LIN {X 0,Y 339.06,Z 977.216,A -85,B 0,C 180,E1 15201.009,E2 15201.009} C_VEL
LIN {X 0,Y 338.438,Z 981.844,A -85,B 0,C 180,E1 15198.238,E2 15198.238} C_VEL
LIN {X 0,Y 338.121,Z 984.855,A -85,B 0,C 180,E1 15195.268,E2 15195.268} C_VEL
LIN {X 0,Y 338.142,Z 986.085,A -85,B 0,C 180,E1 15192.269,E2 15192.269} C_VEL
LIN {X 0,Y 338.465,Z 985.515,A -85,B 0,C 180,E1 15189.419,E2 15189.419} C_VEL
LIN {X 0,Y 339.2,Z 983.049,A -85,B 0,C 180,E1 15186.367,E2 15186.367} C_VEL
LIN {X 0,Y 340.341,Z 978.866,A -85,B 0,C 180,E1 15183.478,E2 15183.478} C_VEL
LIN {X 0,Y 341.875,Z 973.019,A -85,B 0,C 180,E1 15180.764,E2 15180.764} C_VEL
LIN {X 0,Y 343.946,Z 965.145,A -85,B 0,C 180,E1 15178.057,E2 15178.057} C_VEL
LIN {X 0,Y 346.224,Z 956.156,A -85,B 0,C 180,E1 15175.685,E2 15175.685} C_VEL
LIN {X 0,Y 348.825,Z 945.138,A -85,B 0,C 180,E1 15173.402,E2 15173.402} C_VEL
LIN {X 0,Y 351.492,Z 932.886,A -85,B 0,C 180,E1 15171.379,E2 15171.379} C_VEL
LIN {X 0,Y 353.963,Z 920.077,A -85,B 0,C 180,E1 15169.694,E2 15169.694} C_VEL
LIN {X 0,Y 356.266,Z 906.077,A -85,B 0,C 180,E1 15168.227,E2 15168.227} C_VEL
LIN {X 0,Y 358.353,Z 890.745,A -85,B 0,C 180,E1 15166.972,E2 15166.972} C_VEL
LIN {X 0,Y 360,Z 874.678,A -85,B 0,C 180,E1 15165.985,E2 15165.985} C_VEL
LIN {X 0,Y 361.102,Z 857.67,A -85,B 0,C 180,E1 15165.259,E2 15165.259} C_VEL
LIN {X 0,Y 361.863,Z 835.3,A -85,B 0,C 180,E1 15164.69,E2 15164.69} C_VEL
LIN {X 0,Y 365.466,Z 734.296,A -85,B 0,C 180,E1 15162.572,E2 15162.572} C_VEL
LIN {X 0,Y 359.291,Z 705.714,A -85,B 0,C 180,E1 15161.014,E2 15161.014} C_VEL
LIN {X 0,Y 357.272,Z 697.189,A -85,B 0,C 180,E1 15160.487,E2 15160.487} C_VEL
LIN {X 0,Y 358.03,Z 691.708,A -85,B 0,C 180,E1 15159.549,E2 15159.549} C_VEL
LIN {X 0,Y 354.94,Z 678.848,A -85,B 0,C 180,E1 15156.327,E2 15156.327} C_VEL
LIN {X 0,Y 351.349,Z 666.673,A -85,B 0,C 180,E1 15152.913,E2 15152.913} C_VEL
LIN {X 0,Y 347.723,Z 656.229,A -85,B 0,C 180,E1 15149.642,E2 15149.642} C_VEL
LIN {X 0,Y 344.373,Z 647.376,A -85,B 0,C 180,E1 15146.56,E2 15146.56} C_VEL
LIN {X 0,Y 341.041,Z 639.591,A -85,B 0,C 180,E1 15143.499,E2 15143.499} C_VEL
LIN {X 0,Y 339.313,Z 635.632,A -85,B 0,C 180,E1 15141.795,E2 15141.795} C_VEL
LIN {X 0,Y 338.001,Z 632.231,A -85,B 0,C 180,E1 15140.157,E2 15140.157} C_VEL
LIN {X 0,Y 337.989,Z 632.124,A -85,B 0,C 180,E1 15135.793,E2 15135.793} C_VEL
LIN {X 0,Y 337.983,Z 632.122,A -85,B 0,C 180,E1 15131.432,E2 15131.432} C_VEL
LIN {X 0,Y 337.983,Z 632.127,A -85,B 0,C 180,E1 15127.138,E2 15127.138} C_VEL
LIN {X 0,Y 337.978,Z 632.134,A -85,B 0,C 180,E1 15122.713,E2 15122.713} C_VEL
LIN {X 0,Y 337.978,Z 632.135,A -85,B 0,C 180,E1 15118.475,E2 15118.475} C_VEL
LIN {X 0,Y 337.98,Z 632.122,A -85,B 0,C 180,E1 15114.057,E2 15114.057} C_VEL
LIN {X 0,Y 337.978,Z 632.112,A -85,B 0,C 180,E1 15109.776,E2 15109.776} C_VEL
LIN {X 0,Y 337.987,Z 632.108,A -85,B 0,C 180,E1 15105.437,E2 15105.437} C_VEL
LIN {X 0,Y 337.984,Z 632.108,A -85,B 0,C 180,E1 15101.189,E2 15101.189} C_VEL
LIN {X 0,Y 337.988,Z 632.11,A -85,B 0,C 180,E1 15096.928,E2 15096.928} C_VEL
LIN {X 0,Y 337.99,Z 632.112,A -85,B 0,C 180,E1 15092.557,E2 15092.557} C_VEL
LIN {X 0,Y 338.011,Z 632.35,A -85,B 0,C 180,E1 15088.825,E2 15088.825} C_VEL
LIN {X 0,Y 339.689,Z 636.177,A -85,B 0,C 180,E1 15087.208,E2 15087.208} C_VEL
LIN {X 0,Y 342.604,Z 642.181,A -85,B 0,C 180,E1 15084.906,E2 15084.906} C_VEL
LIN {X 0,Y 346.288,Z 649.982,A -85,B 0,C 180,E1 15082.257,E2 15082.257} C_VEL
LIN {X 0,Y 351.256,Z 661.463,A -85,B 0,C 180,E1 15078.887,E2 15078.887} C_VEL
LIN {X 0,Y 356.257,Z 674.185,A -85,B 0,C 180,E1 15075.667,E2 15075.667} C_VEL
LIN {X 0,Y 360.952,Z 687.923,A -85,B 0,C 180,E1 15072.655,E2 15072.655} C_VEL
LIN {X 0,Y 363.777,Z 697.683,A -85,B 0,C 180,E1 15070.762,E2 15070.762} C_VEL
LIN {X 0,Y 362.254,Z 706.393,A -85,B 0,C 180,E1 15069.715,E2 15069.715} C_VEL
LIN {X 0,Y 366.045,Z 739.38,A -85,B 0,C 180,E1 15068.36,E2 15068.36} C_VEL
LIN {X 0,Y 366.683,Z 749.229,A -85,B 0,C 180,E1 15068.034,E2 15068.034} C_VEL
LIN {X 0,Y 361.071,Z 910.999,A -85,B 0,C 180,E1 15064.714,E2 15064.714} C_VEL
LIN {X 0,Y 359.486,Z 930.013,A -85,B 0,C 180,E1 15064.068,E2 15064.068} C_VEL
LIN {X 0,Y 357.3,Z 948.27,A -85,B 0,C 180,E1 15063.167,E2 15063.167} C_VEL
LIN {X 0,Y 354.735,Z 965.817,A -85,B 0,C 180,E1 15061.998,E2 15061.998} C_VEL
LIN {X 0,Y 351.945,Z 982.563,A -85,B 0,C 180,E1 15060.566,E2 15060.566} C_VEL
LIN {X 0,Y 348.905,Z 999.229,A -85,B 0,C 180,E1 15058.779,E2 15058.779} C_VEL
LIN {X 0,Y 345.971,Z 1014.591,A -85,B 0,C 180,E1 15056.746,E2 15056.746} C_VEL
LIN {X 0,Y 343.233,Z 1028.904,A -85,B 0,C 180,E1 15054.434,E2 15054.434} C_VEL
LIN {X 0,Y 340.862,Z 1041.948,A -85,B 0,C 180,E1 15051.871,E2 15051.871} C_VEL
LIN {X 0,Y 338.983,Z 1053.504,A -85,B 0,C 180,E1 15049.111,E2 15049.111} C_VEL
LIN {X 0,Y 337.683,Z 1063.577,A -85,B 0,C 180,E1 15046.16,E2 15046.16} C_VEL
LIN {X 0,Y 336.936,Z 1072.093,A -85,B 0,C 180,E1 15043.034,E2 15043.034} C_VEL
LIN {X 0,Y 336.742,Z 1078.623,A -85,B 0,C 180,E1 15039.916,E2 15039.916} C_VEL
LIN {X 0,Y 336.869,Z 1083.303,A -85,B 0,C 180,E1 15036.818,E2 15036.818} C_VEL
LIN {X 0,Y 337.128,Z 1086.084,A -85,B 0,C 180,E1 15033.911,E2 15033.911} C_VEL
LIN {X 0,Y 337.307,Z 1087.318,A -85,B 0,C 180,E1 15031.019,E2 15031.019} C_VEL
LIN {X 0,Y 337.291,Z 1086.995,A -85,B 0,C 180,E1 15028.131,E2 15028.131} C_VEL
LIN {X 0,Y 337.092,Z 1085.098,A -85,B 0,C 180,E1 15025.236,E2 15025.236} C_VEL
LIN {X 0,Y 336.876,Z 1081.6,A -85,B 0,C 180,E1 15022.324,E2 15022.324} C_VEL
LIN {X 0,Y 336.836,Z 1076.055,A -85,B 0,C 180,E1 15019.221,E2 15019.221} C_VEL
LIN {X 0,Y 337.123,Z 1068.997,A -85,B 0,C 180,E1 15016.274,E2 15016.274} C_VEL
LIN {X 0,Y 337.906,Z 1059.968,A -85,B 0,C 180,E1 15013.32,E2 15013.32} C_VEL
LIN {X 0,Y 339.17,Z 1049.43,A -85,B 0,C 180,E1 15010.541,E2 15010.541} C_VEL
LIN {X 0,Y 340.923,Z 1037.362,A -85,B 0,C 180,E1 15007.935,E2 15007.935} C_VEL
LIN {X 0,Y 343.04,Z 1023.961,A -85,B 0,C 180,E1 15005.55,E2 15005.55} C_VEL
LIN {X 0,Y 345.502,Z 1008.895,A -85,B 0,C 180,E1 15003.348,E2 15003.348} C_VEL
LIN {X 0,Y 348.083,Z 992.738,A -85,B 0,C 180,E1 15001.427,E2 15001.427} C_VEL
LIN {X 0,Y 350.506,Z 976.462,A -85,B 0,C 180,E1 14999.863,E2 14999.863} C_VEL
LIN {X 0,Y 352.865,Z 958.939,A -85,B 0,C 180,E1 14998.528,E2 14998.528} C_VEL
LIN {X 0,Y 354.887,Z 941.144,A -85,B 0,C 180,E1 14997.491,E2 14997.491} C_VEL
LIN {X 0,Y 356.576,Z 922.422,A -85,B 0,C 180,E1 14996.708,E2 14996.708} C_VEL
LIN {X 0,Y 357.533,Z 903.251,A -85,B 0,C 180,E1 14996.184,E2 14996.184} C_VEL
LIN {X 0,Y 361.756,Z 744.837,A -85,B 0,C 180,E1 14993.037,E2 14993.037} C_VEL
LIN {X 0,Y 357.574,Z 706.19,A -85,B 0,C 180,E1 14991.74,E2 14991.74} C_VEL
LIN {X 0,Y 359.524,Z 692.646,A -85,B 0,C 180,E1 14990.136,E2 14990.136} C_VEL
LIN {X 0,Y 352.724,Z 671.714,A -85,B 0,C 180,E1 14986.525,E2 14986.525} C_VEL
LIN {X 0,Y 346.448,Z 654.067,A -85,B 0,C 180,E1 14983.156,E2 14983.156} C_VEL
LIN {X 0,Y 340.366,Z 638.507,A -85,B 0,C 180,E1 14979.821,E2 14979.821} C_VEL
LIN {X 0,Y 338.011,Z 632.324,A -85,B 0,C 180,E1 14978.333,E2 14978.333} C_VEL
LIN {X 0,Y 337.982,Z 632.135,A -85,B 0,C 180,E1 14973.995,E2 14973.995} C_VEL
LIN {X 0,Y 337.983,Z 632.133,A -85,B 0,C 180,E1 14969.606,E2 14969.606} C_VEL
LIN {X 0,Y 338.057,Z 632.553,A -85,B 0,C 180,E1 14968.436,E2 14968.436} C_VEL
LIN {X 0,Y 339.764,Z 636.245,A -85,B 0,C 180,E1 14966.54,E2 14966.54} C_VEL
LIN {X 0,Y 341.678,Z 638.345,A -85,B 0,C 180,E1 14965.279,E2 14965.279} C_VEL
LIN {X 0,Y 343.497,Z 642.043,A -85,B 0,C 180,E1 14963.866,E2 14963.866} C_VEL
LIN {X 0,Y 344.58,Z 643.383,A -85,B 0,C 180,E1 14963.243,E2 14963.243} C_VEL
LIN {X 0,Y 346.37,Z 647.033,A -85,B 0,C 180,E1 14962.041,E2 14962.041} C_VEL
LIN {X 0,Y 347.599,Z 649.52,A -85,B 0,C 180,E1 14961.25,E2 14961.25} C_VEL
LIN {X 0,Y 350.802,Z 655.903,A -85,B 0,C 180,E1 14959.364,E2 14959.364} C_VEL
LIN {X 0,Y 355.065,Z 666.736,A -85,B 0,C 180,E1 14956.692,E2 14956.692} C_VEL
LIN {X 0,Y 358.73,Z 678.676,A -85,B 0,C 180,E1 14954.198,E2 14954.198} C_VEL
LIN {X 0,Y 360.976,Z 688.658,A -85,B 0,C 180,E1 14952.396,E2 14952.396} C_VEL
LIN {X 0,Y 358.887,Z 721.199,A -85,B 0,C 180,E1 14948.168,E2 14948.168} C_VEL
LIN {X 0,Y 358.218,Z 732.321,A -85,B 0,C 180,E1 14946.732,E2 14946.732} C_VEL
LIN {X 0,Y 358.535,Z 735.583,A -85,B 0,C 180,E1 14946.565,E2 14946.565} C_VEL
LIN {X 0,Y 352.855,Z 854.075,A -85,B 0,C 180,E1 14943.431,E2 14943.431} C_VEL
LIN {X 0,Y 352.493,Z 875.546,A -85,B 0,C 180,E1 14942.738,E2 14942.738} C_VEL
LIN {X 0,Y 351.827,Z 891.764,A -85,B 0,C 180,E1 14941.913,E2 14941.913} C_VEL
LIN {X 0,Y 350.744,Z 907.125,A -85,B 0,C 180,E1 14940.816,E2 14940.816} C_VEL
LIN {X 0,Y 349.412,Z 921.154,A -85,B 0,C 180,E1 14939.508,E2 14939.508} C_VEL
LIN {X 0,Y 347.756,Z 934.828,A -85,B 0,C 180,E1 14937.858,E2 14937.858} C_VEL
LIN {X 0,Y 346.179,Z 945.869,A -85,B 0,C 180,E1 14936.191,E2 14936.191} C_VEL
LIN {X 0,Y 344.311,Z 957.347,A -85,B 0,C 180,E1 14933.999,E2 14933.999} C_VEL
LIN {X 0,Y 342.809,Z 965.806,A -85,B 0,C 180,E1 14931.952,E2 14931.952} C_VEL
LIN {X 0,Y 341.337,Z 973.497,A -85,B 0,C 180,E1 14929.536,E2 14929.536} C_VEL
LIN {X 0,Y 340.184,Z 979.292,A -85,B 0,C 180,E1 14927.092,E2 14927.092} C_VEL
LIN {X 0,Y 339.247,Z 983.56,A -85,B 0,C 180,E1 14924.442,E2 14924.442} C_VEL
LIN {X 0,Y 338.625,Z 986.022,A -85,B 0,C 180,E1 14921.76,E2 14921.76} C_VEL
LIN {X 0,Y 338.262,Z 986.646,A -85,B 0,C 180,E1 14919.043,E2 14919.043} C_VEL
LIN {X 0,Y 338.137,Z 985.591,A -85,B 0,C 180,E1 14916.444,E2 14916.444} C_VEL
LIN {X 0,Y 338.224,Z 982.594,A -85,B 0,C 180,E1 14913.677,E2 14913.677} C_VEL
LIN {X 0,Y 338.562,Z 977.934,A -85,B 0,C 180,E1 14911.031,E2 14911.031} C_VEL
LIN {X 0,Y 339.183,Z 971.133,A -85,B 0,C 180,E1 14908.35,E2 14908.35} C_VEL
LIN {X 0,Y 339.976,Z 963.349,A -85,B 0,C 180,E1 14906.028,E2 14906.028} C_VEL
LIN {X 0,Y 341.057,Z 953.317,A -85,B 0,C 180,E1 14903.687,E2 14903.687} C_VEL
LIN {X 0,Y 342.233,Z 942.324,A -85,B 0,C 180,E1 14901.649,E2 14901.649} C_VEL
LIN {X 0,Y 343.534,Z 929.537,A -85,B 0,C 180,E1 14899.749,E2 14899.749} C_VEL
LIN {X 0,Y 344.73,Z 916.049,A -85,B 0,C 180,E1 14898.156,E2 14898.156} C_VEL
LIN {X 0,Y 345.875,Z 901.008,A -85,B 0,C 180,E1 14896.754,E2 14896.754} C_VEL
LIN {X 0,Y 346.777,Z 885.221,A -85,B 0,C 180,E1 14895.649,E2 14895.649} C_VEL
LIN {X 0,Y 347.396,Z 868.788,A -85,B 0,C 180,E1 14894.82,E2 14894.82} C_VEL
LIN {X 0,Y 347.674,Z 849.904,A -85,B 0,C 180,E1 14894.232,E2 14894.232} C_VEL
LIN {X 0,Y 351.149,Z 727.334,A -85,B 0,C 180,E1 14891.298,E2 14891.298} C_VEL
LIN {X 0,Y 349.786,Z 718.722,A -85,B 0,C 180,E1 14890.944,E2 14890.944} C_VEL
LIN {X 0,Y 351.327,Z 685.759,A -85,B 0,C 180,E1 14886.624,E2 14886.624} C_VEL
LIN {X 0,Y 351.501,Z 677.083,A -85,B 0,C 180,E1 14885.471,E2 14885.471} C_VEL
LIN {X 0,Y 346.652,Z 658.977,A -85,B 0,C 180,E1 14882.543,E2 14882.543} C_VEL
LIN {X 0,Y 340.965,Z 641.141,A -85,B 0,C 180,E1 14879.515,E2 14879.515} C_VEL
LIN {X 0,Y 337.99,Z 632.399,A -85,B 0,C 180,E1 14877.914,E2 14877.914} C_VEL
LIN {X 0,Y 338.002,Z 632.326,A -85,B 0,C 180,E1 14877.196,E2 14877.196} C_VEL
LIN {X 0,Y 342.322,Z 645.106,A -85,B 0,C 180,E1 14873.771,E2 14873.771} C_VEL
LIN {X 0,Y 346.804,Z 659.68,A -85,B 0,C 180,E1 14870.241,E2 14870.241} C_VEL
LIN {X 0,Y 350.837,Z 675.127,A -85,B 0,C 180,E1 14866.748,E2 14866.748} C_VEL
LIN {X 0,Y 352.481,Z 682.884,A -85,B 0,C 180,E1 14865.128,E2 14865.128} C_VEL
LIN {X 0,Y 350.755,Z 696.336,A -85,B 0,C 180,E1 14862.862,E2 14862.862} C_VEL
LIN {X 0,Y 357.513,Z 732.878,A -85,B 0,C 180,E1 14861.392,E2 14861.392} C_VEL
LIN {X 0,Y 355.604,Z 799.245,A -85,B 0,C 180,E1 14860.057,E2 14860.057} C_VEL
LIN {X 0,Y 354.5,Z 806.914,A -85,B 0,C 180,E1 14859.975,E2 14859.975} C_VEL
LIN {X 0,Y 348.365,Z 827.251,A -85,B 0,C 180,E1 14860.018,E2 14860.018} C_VEL
LIN {X 0,Y 347.475,Z 833.835,A -85,B 0,C 180,E1 14859.938,E2 14859.938} C_VEL
LIN {X 0,Y 346.865,Z 856.618,A -85,B 0,C 180,E1 14859.358,E2 14859.358} C_VEL
LIN {X 0,Y 345.99,Z 873.229,A -85,B 0,C 180,E1 14858.643,E2 14858.643} C_VEL
LIN {X 0,Y 344.7,Z 888.944,A -85,B 0,C 180,E1 14857.668,E2 14857.668} C_VEL
LIN {X 0,Y 342.989,Z 904.766,A -85,B 0,C 180,E1 14856.36,E2 14856.36} C_VEL
LIN {X 0,Y 341.053,Z 919.501,A -85,B 0,C 180,E1 14854.793,E2 14854.793} C_VEL
LIN {X 0,Y 338.999,Z 933.03,A -85,B 0,C 180,E1 14852.959,E2 14852.959} C_VEL
LIN {X 0,Y 336.929,Z 945.502,A -85,B 0,C 180,E1 14850.851,E2 14850.851} C_VEL
LIN {X 0,Y 335.054,Z 956.083,A -85,B 0,C 180,E1 14848.613,E2 14848.613} C_VEL
LIN {X 0,Y 333.321,Z 965.671,A -85,B 0,C 180,E1 14846.044,E2 14846.044} C_VEL
LIN {X 0,Y 332.009,Z 973.276,A -85,B 0,C 180,E1 14843.429,E2 14843.429} C_VEL
LIN {X 0,Y 331.032,Z 979.374,A -85,B 0,C 180,E1 14840.613,E2 14840.613} C_VEL
LIN {X 0,Y 330.417,Z 983.875,A -85,B 0,C 180,E1 14837.594,E2 14837.594} C_VEL
LIN {X 0,Y 330.186,Z 986.413,A -85,B 0,C 180,E1 14834.726,E2 14834.726} C_VEL
LIN {X 0,Y 330.258,Z 987.292,A -85,B 0,C 180,E1 14831.831,E2 14831.831} C_VEL
LIN {X 0,Y 330.692,Z 986.44,A -85,B 0,C 180,E1 14828.727,E2 14828.727} C_VEL
LIN {X 0,Y 331.509,Z 983.916,A -85,B 0,C 180,E1 14825.784,E2 14825.784} C_VEL
LIN {X 0,Y 332.783,Z 979.475,A -85,B 0,C 180,E1 14822.827,E2 14822.827} C_VEL
LIN {X 0,Y 334.493,Z 973.448,A -85,B 0,C 180,E1 14820.054,E2 14820.054} C_VEL
LIN {X 0,Y 336.591,Z 965.964,A -85,B 0,C 180,E1 14817.475,E2 14817.475} C_VEL
LIN {X 0,Y 338.994,Z 956.974,A -85,B 0,C 180,E1 14815.081,E2 14815.081} C_VEL
LIN {X 0,Y 341.676,Z 946.259,A -85,B 0,C 180,E1 14812.823,E2 14812.823} C_VEL
LIN {X 0,Y 344.51,Z 933.947,A -85,B 0,C 180,E1 14810.751,E2 14810.751} C_VEL
LIN {X 0,Y 347.226,Z 920.511,A -85,B 0,C 180,E1 14808.964,E2 14808.964} C_VEL
LIN {X 0,Y 349.742,Z 905.838,A -85,B 0,C 180,E1 14807.423,E2 14807.423} C_VEL
LIN {X 0,Y 351.848,Z 890.928,A -85,B 0,C 180,E1 14806.204,E2 14806.204} C_VEL
LIN {X 0,Y 353.544,Z 874.739,A -85,B 0,C 180,E1 14805.212,E2 14805.212} C_VEL
LIN {X 0,Y 354.7,Z 857.424,A -85,B 0,C 180,E1 14804.478,E2 14804.478} C_VEL
LIN {X 0,Y 355.575,Z 832.802,A -85,B 0,C 180,E1 14803.863,E2 14803.863} C_VEL
LIN {X 0,Y 359.215,Z 735.783,A -85,B 0,C 180,E1 14801.795,E2 14801.795} C_VEL
LIN {X 0,Y 353.238,Z 707.82,A -85,B 0,C 180,E1 14800.22,E2 14800.22} C_VEL
LIN {X 0,Y 350.81,Z 697.556,A -85,B 0,C 180,E1 14799.57,E2 14799.57} C_VEL
LIN {X 0,Y 351.012,Z 694.769,A -85,B 0,C 180,E1 14799.12,E2 14799.12} C_VEL
LIN {X 0,Y 348.024,Z 682.157,A -85,B 0,C 180,E1 14795.88,E2 14795.88} C_VEL
LIN {X 0,Y 344.438,Z 669.949,A -85,B 0,C 180,E1 14792.357,E2 14792.357} C_VEL
LIN {X 0,Y 340.714,Z 658.978,A -85,B 0,C 180,E1 14788.769,E2 14788.769} C_VEL
LIN {X 0,Y 336.874,Z 649.01,A -85,B 0,C 180,E1 14785.115,E2 14785.115} C_VEL
LIN {X 0,Y 333.589,Z 641.25,A -85,B 0,C 180,E1 14781.819,E2 14781.819} C_VEL
LIN {X 0,Y 331.37,Z 636.624,A -85,B 0,C 180,E1 14779.568,E2 14779.568} C_VEL
LIN {X 0,Y 330.058,Z 633.196,A -85,B 0,C 180,E1 14777.725,E2 14777.725} C_VEL
LIN {X 0,Y 330.043,Z 633.107,A -85,B 0,C 180,E1 14773.312,E2 14773.312} C_VEL
LIN {X 0,Y 330.041,Z 633.107,A -85,B 0,C 180,E1 14768.888,E2 14768.888} C_VEL
LIN {X 0,Y 330.039,Z 633.103,A -85,B 0,C 180,E1 14764.518,E2 14764.518} C_VEL
LIN {X 0,Y 330.046,Z 633.096,A -85,B 0,C 180,E1 14760.174,E2 14760.174} C_VEL
LIN {X 0,Y 330.043,Z 633.092,A -85,B 0,C 180,E1 14755.831,E2 14755.831} C_VEL
LIN {X 0,Y 330.051,Z 633.094,A -85,B 0,C 180,E1 14751.464,E2 14751.464} C_VEL
LIN {X 0,Y 330.05,Z 633.101,A -85,B 0,C 180,E1 14747.046,E2 14747.046} C_VEL
LIN {X 0,Y 330.05,Z 633.109,A -85,B 0,C 180,E1 14742.73,E2 14742.73} C_VEL
LIN {X 0,Y 330.057,Z 633.111,A -85,B 0,C 180,E1 14738.31,E2 14738.31} C_VEL
LIN {X 0,Y 330.042,Z 633.112,A -85,B 0,C 180,E1 14733.943,E2 14733.943} C_VEL
LIN {X 0,Y 330.077,Z 633.401,A -85,B 0,C 180,E1 14731.208,E2 14731.208} C_VEL
LIN {X 0,Y 331.809,Z 637.228,A -85,B 0,C 180,E1 14729.386,E2 14729.386} C_VEL
LIN {X 0,Y 334.901,Z 643.522,A -85,B 0,C 180,E1 14726.714,E2 14726.714} C_VEL
LIN {X 0,Y 337.164,Z 648.364,A -85,B 0,C 180,E1 14724.879,E2 14724.879} C_VEL
LIN {X 0,Y 340.426,Z 655.31,A -85,B 0,C 180,E1 14722.467,E2 14722.467} C_VEL
LIN {X 0,Y 345.198,Z 666.52,A -85,B 0,C 180,E1 14719.111,E2 14719.111} C_VEL
LIN {X 0,Y 350.184,Z 679.483,A -85,B 0,C 180,E1 14715.779,E2 14715.779} C_VEL
LIN {X 0,Y 354.645,Z 692.9,A -85,B 0,C 180,E1 14712.801,E2 14712.801} C_VEL
LIN {X 0,Y 356.783,Z 701.131,A -85,B 0,C 180,E1 14711.191,E2 14711.191} C_VEL
LIN {X 0,Y 355.883,Z 706.598,A -85,B 0,C 180,E1 14710.556,E2 14710.556} C_VEL
LIN {X 0,Y 359.68,Z 739.617,A -85,B 0,C 180,E1 14709.158,E2 14709.158} C_VEL
LIN {X 0,Y 360.363,Z 750.147,A -85,B 0,C 180,E1 14708.798,E2 14708.798} C_VEL
LIN {X 0,Y 354.502,Z 910.191,A -85,B 0,C 180,E1 14705.459,E2 14705.459} C_VEL
LIN {X 0,Y 352.858,Z 929.149,A -85,B 0,C 180,E1 14704.805,E2 14704.805} C_VEL
LIN {X 0,Y 350.586,Z 947.347,A -85,B 0,C 180,E1 14703.897,E2 14703.897} C_VEL
LIN {X 0,Y 347.883,Z 964.988,A -85,B 0,C 180,E1 14702.706,E2 14702.706} C_VEL
LIN {X 0,Y 344.801,Z 982.527,A -85,B 0,C 180,E1 14701.172,E2 14701.172} C_VEL
LIN {X 0,Y 341.623,Z 999.001,A -85,B 0,C 180,E1 14699.356,E2 14699.356} C_VEL
LIN {X 0,Y 338.493,Z 1014.448,A -85,B 0,C 180,E1 14697.248,E2 14697.248} C_VEL
LIN {X 0,Y 335.567,Z 1028.854,A -85,B 0,C 180,E1 14694.842,E2 14694.842} C_VEL
LIN {X 0,Y 333.083,Z 1041.723,A -85,B 0,C 180,E1 14692.224,E2 14692.224} C_VEL
LIN {X 0,Y 331.109,Z 1053.112,A -85,B 0,C 180,E1 14689.4,E2 14689.4} C_VEL
LIN {X 0,Y 329.745,Z 1063.021,A -85,B 0,C 180,E1 14686.379,E2 14686.379} C_VEL
LIN {X 0,Y 328.965,Z 1071.377,A -85,B 0,C 180,E1 14683.176,E2 14683.176} C_VEL
LIN {X 0,Y 328.772,Z 1077.784,A -85,B 0,C 180,E1 14679.982,E2 14679.982} C_VEL
LIN {X 0,Y 328.921,Z 1082.359,A -85,B 0,C 180,E1 14676.808,E2 14676.808} C_VEL
LIN {X 0,Y 329.206,Z 1085.05,A -85,B 0,C 180,E1 14673.831,E2 14673.831} C_VEL
LIN {X 0,Y 329.398,Z 1086.161,A -85,B 0,C 180,E1 14670.869,E2 14670.869} C_VEL
LIN {X 0,Y 329.369,Z 1085.704,A -85,B 0,C 180,E1 14667.912,E2 14667.912} C_VEL
LIN {X 0,Y 329.149,Z 1083.662,A -85,B 0,C 180,E1 14664.946,E2 14664.946} C_VEL
LIN {X 0,Y 328.921,Z 1080.004,A -85,B 0,C 180,E1 14661.961,E2 14661.961} C_VEL
LIN {X 0,Y 328.886,Z 1074.661,A -85,B 0,C 180,E1 14658.958,E2 14658.958} C_VEL
LIN {X 0,Y 329.204,Z 1067.522,A -85,B 0,C 180,E1 14655.937,E2 14655.937} C_VEL
LIN {X 0,Y 330.049,Z 1058.407,A -85,B 0,C 180,E1 14652.911,E2 14652.911} C_VEL
LIN {X 0,Y 331.412,Z 1047.772,A -85,B 0,C 180,E1 14650.067,E2 14650.067} C_VEL
LIN {X 0,Y 333.264,Z 1035.649,A -85,B 0,C 180,E1 14647.416,E2 14647.416} C_VEL
LIN {X 0,Y 335.556,Z 1021.819,A -85,B 0,C 180,E1 14644.935,E2 14644.935} C_VEL
LIN {X 0,Y 338.123,Z 1006.733,A -85,B 0,C 180,E1 14642.719,E2 14642.719} C_VEL
LIN {X 0,Y 340.717,Z 991.112,A -85,B 0,C 180,E1 14640.847,E2 14640.847} C_VEL
LIN {X 0,Y 343.301,Z 974.352,A -85,B 0,C 180,E1 14639.225,E2 14639.225} C_VEL
LIN {X 0,Y 345.786,Z 956.362,A -85,B 0,C 180,E1 14637.856,E2 14637.856} C_VEL
LIN {X 0,Y 347.903,Z 938.054,A -85,B 0,C 180,E1 14636.804,E2 14636.804} C_VEL
LIN {X 0,Y 349.606,Z 918.728,A -85,B 0,C 180,E1 14636.027,E2 14636.027} C_VEL
LIN {X 0,Y 350.497,Z 898.279,A -85,B 0,C 180,E1 14635.51,E2 14635.51} C_VEL
LIN {X 0,Y 354.741,Z 745.778,A -85,B 0,C 180,E1 14632.433,E2 14632.433} C_VEL
LIN {X 0,Y 350.512,Z 706.051,A -85,B 0,C 180,E1 14631.076,E2 14631.076} C_VEL
LIN {X 0,Y 352.198,Z 695.332,A -85,B 0,C 180,E1 14629.788,E2 14629.788} C_VEL
LIN {X 0,Y 345.483,Z 674.47,A -85,B 0,C 180,E1 14626.106,E2 14626.106} C_VEL
LIN {X 0,Y 339.313,Z 657.007,A -85,B 0,C 180,E1 14622.667,E2 14622.667} C_VEL
LIN {X 0,Y 333.623,Z 642.41,A -85,B 0,C 180,E1 14619.446,E2 14619.446} C_VEL
LIN {X 0,Y 330.638,Z 635.288,A -85,B 0,C 180,E1 14617.706,E2 14617.706} C_VEL
LIN {X 0,Y 330.399,Z 634.661,A -85,B 0,C 180,E1 14616.972,E2 14616.972} C_VEL
LIN {X 0,Y 330.457,Z 634.833,A -85,B 0,C 180,E1 14614.614,E2 14614.614} C_VEL
LIN {X 0,Y 332.236,Z 637.684,A -85,B 0,C 180,E1 14610.57,E2 14610.57} C_VEL
LIN {X 0,Y 334.164,Z 639.508,A -85,B 0,C 180,E1 14608.603,E2 14608.603} C_VEL
LIN {X 0,Y 335.862,Z 643.154,A -85,B 0,C 180,E1 14606.713,E2 14606.713} C_VEL
LIN {X 0,Y 337.409,Z 644.799,A -85,B 0,C 180,E1 14605.635,E2 14605.635} C_VEL
LIN {X 0,Y 339.05,Z 648.449,A -85,B 0,C 180,E1 14604.199,E2 14604.199} C_VEL
LIN {X 0,Y 340.163,Z 650.003,A -85,B 0,C 180,E1 14603.496,E2 14603.496} C_VEL
LIN {X 0,Y 342.86,Z 655.778,A -85,B 0,C 180,E1 14601.52,E2 14601.52} C_VEL
LIN {X 0,Y 345.615,Z 661.467,A -85,B 0,C 180,E1 14599.784,E2 14599.784} C_VEL
LIN {X 0,Y 349.515,Z 671.818,A -85,B 0,C 180,E1 14597.136,E2 14597.136} C_VEL
LIN {X 0,Y 352.87,Z 683.211,A -85,B 0,C 180,E1 14594.69,E2 14594.69} C_VEL
LIN {X 0,Y 354.767,Z 692.519,A -85,B 0,C 180,E1 14592.947,E2 14592.947} C_VEL
LIN {X 0,Y 352.566,Z 723.35,A -85,B 0,C 180,E1 14588.891,E2 14588.891} C_VEL
LIN {X 0,Y 351.956,Z 734.54,A -85,B 0,C 180,E1 14587.462,E2 14587.462} C_VEL
LIN {X 0,Y 352.195,Z 737.348,A -85,B 0,C 180,E1 14587.329,E2 14587.329} C_VEL
LIN {X 0,Y 346.058,Z 856.501,A -85,B 0,C 180,E1 14584.074,E2 14584.074} C_VEL
LIN {X 0,Y 345.657,Z 877.48,A -85,B 0,C 180,E1 14583.368,E2 14583.368} C_VEL
LIN {X 0,Y 344.945,Z 893.445,A -85,B 0,C 180,E1 14582.533,E2 14582.533} C_VEL
LIN {X 0,Y 343.783,Z 908.674,A -85,B 0,C 180,E1 14581.416,E2 14581.416} C_VEL
LIN {X 0,Y 342.352,Z 922.6,A -85,B 0,C 180,E1 14580.083,E2 14580.083} C_VEL
LIN {X 0,Y 340.504,Z 936.855,A -85,B 0,C 180,E1 14578.317,E2 14578.317} C_VEL
LIN {X 0,Y 338.829,Z 947.772,A -85,B 0,C 180,E1 14576.616,E2 14576.616} C_VEL
LIN {X 0,Y 336.985,Z 958.338,A -85,B 0,C 180,E1 14574.551,E2 14574.551} C_VEL
LIN {X 0,Y 335.236,Z 967.462,A -85,B 0,C 180,E1 14572.286,E2 14572.286} C_VEL
LIN {X 0,Y 333.672,Z 975.093,A -85,B 0,C 180,E1 14569.816,E2 14569.816} C_VEL
LIN {X 0,Y 332.436,Z 980.804,A -85,B 0,C 180,E1 14567.316,E2 14567.316} C_VEL
LIN {X 0,Y 331.43,Z 984.992,A -85,B 0,C 180,E1 14564.604,E2 14564.604} C_VEL
LIN {X 0,Y 330.793,Z 987.266,A -85,B 0,C 180,E1 14562.042,E2 14562.042} C_VEL
LIN {X 0,Y 330.38,Z 987.916,A -85,B 0,C 180,E1 14559.255,E2 14559.255} C_VEL
LIN {X 0,Y 330.225,Z 986.778,A -85,B 0,C 180,E1 14556.442,E2 14556.442} C_VEL
LIN {X 0,Y 330.314,Z 983.664,A -85,B 0,C 180,E1 14553.578,E2 14553.578} C_VEL
LIN {X 0,Y 330.667,Z 978.873,A -85,B 0,C 180,E1 14550.867,E2 14550.867} C_VEL
LIN {X 0,Y 331.325,Z 971.964,A -85,B 0,C 180,E1 14548.122,E2 14548.122} C_VEL
LIN {X 0,Y 332.159,Z 964.022,A -85,B 0,C 180,E1 14545.743,E2 14545.743} C_VEL
LIN {X 0,Y 333.302,Z 953.853,A -85,B 0,C 180,E1 14543.346,E2 14543.346} C_VEL
LIN {X 0,Y 334.529,Z 942.7,A -85,B 0,C 180,E1 14541.27,E2 14541.27} C_VEL
LIN {X 0,Y 335.846,Z 930.206,A -85,B 0,C 180,E1 14539.392,E2 14539.392} C_VEL
LIN {X 0,Y 337.154,Z 915.833,A -85,B 0,C 180,E1 14537.686,E2 14537.686} C_VEL
LIN {X 0,Y 338.301,Z 901.016,A -85,B 0,C 180,E1 14536.307,E2 14536.307} C_VEL
LIN {X 0,Y 339.277,Z 884.325,A -85,B 0,C 180,E1 14535.141,E2 14535.141} C_VEL
LIN {X 0,Y 339.872,Z 867.676,A -85,B 0,C 180,E1 14534.329,E2 14534.329} C_VEL
LIN {X 0,Y 340.161,Z 848.179,A -85,B 0,C 180,E1 14533.739,E2 14533.739} C_VEL
LIN {X 0,Y 343.78,Z 728.437,A -85,B 0,C 180,E1 14530.799,E2 14530.799} C_VEL
LIN {X 0,Y 342.422,Z 719.479,A -85,B 0,C 180,E1 14530.409,E2 14530.409} C_VEL
LIN {X 0,Y 344.04,Z 686.509,A -85,B 0,C 180,E1 14526.052,E2 14526.052} C_VEL
LIN {X 0,Y 344.173,Z 679.617,A -85,B 0,C 180,E1 14525.115,E2 14525.115} C_VEL
LIN {X 0,Y 339.435,Z 661.905,A -85,B 0,C 180,E1 14522.22,E2 14522.22} C_VEL
LIN {X 0,Y 333.895,Z 644.484,A -85,B 0,C 180,E1 14519.217,E2 14519.217} C_VEL
LIN {X 0,Y 331.044,Z 636.184,A -85,B 0,C 180,E1 14517.67,E2 14517.67} C_VEL
LIN {X 0,Y 331.094,Z 636.244,A -85,B 0,C 180,E1 14517.396,E2 14517.396} C_VEL
LIN {X 0,Y 335.545,Z 649.436,A -85,B 0,C 180,E1 14513.822,E2 14513.822} C_VEL
LIN {X 0,Y 339.942,Z 664.059,A -85,B 0,C 180,E1 14510.237,E2 14510.237} C_VEL
LIN {X 0,Y 343.838,Z 679.293,A -85,B 0,C 180,E1 14506.732,E2 14506.732} C_VEL
LIN {X 0,Y 345.053,Z 685.202,A -85,B 0,C 180,E1 14505.462,E2 14505.462} C_VEL
LIN {X 0,Y 343.564,Z 696.202,A -85,B 0,C 180,E1 14503.582,E2 14503.582} C_VEL
LIN {X 0,Y 350.487,Z 734.043,A -85,B 0,C 180,E1 14502,E2 14502} C_VEL
LIN {X 0,Y 347.475,Z 833.835,A -85,B 0,C 180,E1 14499.938,E2 14499.938} C_VEL
LIN {X 0,Y 346.368,Z 841.519,A -85,B 0,C 180,E1 14499.851,E2 14499.851} C_VEL
LIN {X 0,Y 340.779,Z 859.672,A -85,B 0,C 180,E1 14499.776,E2 14499.776} C_VEL
LIN {X 0,Y 339.278,Z 867.151,A -85,B 0,C 180,E1 14499.558,E2 14499.558} C_VEL
LIN {X 0,Y 339.183,Z 868.214,A -85,B 0,C 180,E1 14499.508,E2 14499.508} C_VEL
LIN {X 0,Y 337.962,Z 884.433,A -85,B 0,C 180,E1 14498.593,E2 14498.593} C_VEL
LIN {X 0,Y 336.284,Z 900.71,A -85,B 0,C 180,E1 14497.346,E2 14497.346} C_VEL
LIN {X 0,Y 334.329,Z 915.704,A -85,B 0,C 180,E1 14495.836,E2 14495.836} C_VEL
LIN {X 0,Y 332.124,Z 930.238,A -85,B 0,C 180,E1 14493.971,E2 14493.971} C_VEL
LIN {X 0,Y 330.14,Z 942.031,A -85,B 0,C 180,E1 14492.083,E2 14492.083} C_VEL
LIN {X 0,Y 328.071,Z 953.357,A -85,B 0,C 180,E1 14489.826,E2 14489.826} C_VEL
LIN {X 0,Y 326.217,Z 963.214,A -85,B 0,C 180,E1 14487.365,E2 14487.365} C_VEL
LIN {X 0,Y 324.672,Z 971.629,A -85,B 0,C 180,E1 14484.699,E2 14484.699} C_VEL
LIN {X 0,Y 323.479,Z 978.442,A -85,B 0,C 180,E1 14481.826,E2 14481.826} C_VEL
LIN {X 0,Y 322.724,Z 983.409,A -85,B 0,C 180,E1 14478.926,E2 14478.926} C_VEL
LIN {X 0,Y 322.34,Z 986.685,A -85,B 0,C 180,E1 14475.999,E2 14475.999} C_VEL
LIN {X 0,Y 322.278,Z 988.289,A -85,B 0,C 180,E1 14473.045,E2 14473.045} C_VEL
LIN {X 0,Y 322.577,Z 988.229,A -85,B 0,C 180,E1 14469.876,E2 14469.876} C_VEL
LIN {X 0,Y 323.314,Z 986.358,A -85,B 0,C 180,E1 14466.706,E2 14466.706} C_VEL
LIN {X 0,Y 324.484,Z 982.646,A -85,B 0,C 180,E1 14463.659,E2 14463.659} C_VEL
LIN {X 0,Y 326.213,Z 977.026,A -85,B 0,C 180,E1 14460.633,E2 14460.633} C_VEL
LIN {X 0,Y 328.249,Z 970.287,A -85,B 0,C 180,E1 14457.994,E2 14457.994} C_VEL
LIN {X 0,Y 330.789,Z 961.466,A -85,B 0,C 180,E1 14455.372,E2 14455.372} C_VEL
LIN {X 0,Y 333.613,Z 951.118,A -85,B 0,C 180,E1 14452.958,E2 14452.958} C_VEL
LIN {X 0,Y 336.451,Z 939.847,A -85,B 0,C 180,E1 14450.863,E2 14450.863} C_VEL
LIN {X 0,Y 339.374,Z 926.724,A -85,B 0,C 180,E1 14448.929,E2 14448.929} C_VEL
LIN {X 0,Y 342.058,Z 912.851,A -85,B 0,C 180,E1 14447.301,E2 14447.301} C_VEL
LIN {X 0,Y 344.431,Z 898.287,A -85,B 0,C 180,E1 14445.953,E2 14445.953} C_VEL
LIN {X 0,Y 346.441,Z 882.261,A -85,B 0,C 180,E1 14444.826,E2 14444.826} C_VEL
LIN {X 0,Y 347.94,Z 864.923,A -85,B 0,C 180,E1 14443.951,E2 14443.951} C_VEL
LIN {X 0,Y 348.757,Z 847.699,A -85,B 0,C 180,E1 14443.392,E2 14443.392} C_VEL
LIN {X 0,Y 353.053,Z 737.354,A -85,B 0,C 180,E1 14440.994,E2 14440.994} C_VEL
LIN {X 0,Y 347.065,Z 709.017,A -85,B 0,C 180,E1 14439.345,E2 14439.345} C_VEL
LIN {X 0,Y 344.25,Z 698.024,A -85,B 0,C 180,E1 14438.59,E2 14438.59} C_VEL
LIN {X 0,Y 343.531,Z 695.564,A -85,B 0,C 180,E1 14438.1,E2 14438.1} C_VEL
LIN {X 0,Y 340.639,Z 683.716,A -85,B 0,C 180,E1 14434.916,E2 14434.916} C_VEL
LIN {X 0,Y 337.15,Z 671.92,A -85,B 0,C 180,E1 14431.34,E2 14431.34} C_VEL
LIN {X 0,Y 333.358,Z 660.8,A -85,B 0,C 180,E1 14427.51,E2 14427.51} C_VEL
LIN {X 0,Y 330.008,Z 652.469,A -85,B 0,C 180,E1 14424.222,E2 14424.222} C_VEL
LIN {X 0,Y 327.441,Z 646.242,A -85,B 0,C 180,E1 14421.496,E2 14421.496} C_VEL
LIN {X 0,Y 325.467,Z 641.945,A -85,B 0,C 180,E1 14419.378,E2 14419.378} C_VEL
LIN {X 0,Y 323.672,Z 637.95,A -85,B 0,C 180,E1 14417.251,E2 14417.251} C_VEL
LIN {X 0,Y 322.12,Z 634.204,A -85,B 0,C 180,E1 14414.93,E2 14414.93} C_VEL
LIN {X 0,Y 322.105,Z 634.088,A -85,B 0,C 180,E1 14410.553,E2 14410.553} C_VEL
LIN {X 0,Y 322.111,Z 634.088,A -85,B 0,C 180,E1 14406.237,E2 14406.237} C_VEL
LIN {X 0,Y 322.108,Z 634.09,A -85,B 0,C 180,E1 14401.779,E2 14401.779} C_VEL
LIN {X 0,Y 322.108,Z 634.096,A -85,B 0,C 180,E1 14397.332,E2 14397.332} C_VEL
LIN {X 0,Y 322.118,Z 634.104,A -85,B 0,C 180,E1 14392.868,E2 14392.868} C_VEL
LIN {X 0,Y 322.103,Z 634.112,A -85,B 0,C 180,E1 14388.36,E2 14388.36} C_VEL
LIN {X 0,Y 322.099,Z 634.109,A -85,B 0,C 180,E1 14383.962,E2 14383.962} C_VEL
LIN {X 0,Y 322.101,Z 634.105,A -85,B 0,C 180,E1 14379.466,E2 14379.466} C_VEL
LIN {X 0,Y 322.105,Z 634.107,A -85,B 0,C 180,E1 14375.013,E2 14375.013} C_VEL
LIN {X 0,Y 322.179,Z 634.582,A -85,B 0,C 180,E1 14373.926,E2 14373.926} C_VEL
LIN {X 0,Y 324.013,Z 638.368,A -85,B 0,C 180,E1 14371.827,E2 14371.827} C_VEL
LIN {X 0,Y 327.07,Z 644.506,A -85,B 0,C 180,E1 14368.866,E2 14368.866} C_VEL
LIN {X 0,Y 329.324,Z 649.23,A -85,B 0,C 180,E1 14366.873,E2 14366.873} C_VEL
LIN {X 0,Y 332.76,Z 656.39,A -85,B 0,C 180,E1 14364.132,E2 14364.132} C_VEL
LIN {X 0,Y 337.637,Z 667.766,A -85,B 0,C 180,E1 14360.455,E2 14360.455} C_VEL
LIN {X 0,Y 342.36,Z 679.869,A -85,B 0,C 180,E1 14357.12,E2 14357.12} C_VEL
LIN {X 0,Y 346.965,Z 693.394,A -85,B 0,C 180,E1 14353.91,E2 14353.91} C_VEL
LIN {X 0,Y 349.946,Z 703.817,A -85,B 0,C 180,E1 14351.737,E2 14351.737} C_VEL
LIN {X 0,Y 349.645,Z 707.017,A -85,B 0,C 180,E1 14351.423,E2 14351.423} C_VEL
LIN {X 0,Y 353.343,Z 739.255,A -85,B 0,C 180,E1 14350.015,E2 14350.015} C_VEL
LIN {X 0,Y 354.113,Z 751.26,A -85,B 0,C 180,E1 14349.587,E2 14349.587} C_VEL
LIN {X 0,Y 348.033,Z 909.268,A -85,B 0,C 180,E1 14346.241,E2 14346.241} C_VEL
LIN {X 0,Y 346.329,Z 928.265,A -85,B 0,C 180,E1 14345.579,E2 14345.579} C_VEL
LIN {X 0,Y 343.98,Z 946.239,A -85,B 0,C 180,E1 14344.672,E2 14344.672} C_VEL
LIN {X 0,Y 341.275,Z 963.197,A -85,B 0,C 180,E1 14343.522,E2 14343.522} C_VEL
LIN {X 0,Y 338.181,Z 980.026,A -85,B 0,C 180,E1 14342.053,E2 14342.053} C_VEL
LIN {X 0,Y 334.874,Z 996.449,A -85,B 0,C 180,E1 14340.248,E2 14340.248} C_VEL
LIN {X 0,Y 331.591,Z 1011.81,A -85,B 0,C 180,E1 14338.157,E2 14338.157} C_VEL
LIN {X 0,Y 328.521,Z 1025.965,A -85,B 0,C 180,E1 14335.799,E2 14335.799} C_VEL
LIN {X 0,Y 325.785,Z 1039.09,A -85,B 0,C 180,E1 14333.131,E2 14333.131} C_VEL
LIN {X 0,Y 323.578,Z 1050.715,A -85,B 0,C 180,E1 14330.247,E2 14330.247} C_VEL
LIN {X 0,Y 322.009,Z 1060.852,A -85,B 0,C 180,E1 14327.156,E2 14327.156} C_VEL
LIN {X 0,Y 321.12,Z 1068.995,A -85,B 0,C 180,E1 14324.055,E2 14324.055} C_VEL
LIN {X 0,Y 320.809,Z 1075.698,A -85,B 0,C 180,E1 14320.777,E2 14320.777} C_VEL
LIN {X 0,Y 320.918,Z 1080.55,A -85,B 0,C 180,E1 14317.519,E2 14317.519} C_VEL
LIN {X 0,Y 321.217,Z 1083.493,A -85,B 0,C 180,E1 14314.463,E2 14314.463} C_VEL
LIN {X 0,Y 321.464,Z 1084.88,A -85,B 0,C 180,E1 14311.425,E2 14311.425} C_VEL
LIN {X 0,Y 321.482,Z 1084.759,A -85,B 0,C 180,E1 14308.574,E2 14308.574} C_VEL
LIN {X 0,Y 321.274,Z 1083.072,A -85,B 0,C 180,E1 14305.537,E2 14305.537} C_VEL
LIN {X 0,Y 321.01,Z 1079.721,A -85,B 0,C 180,E1 14302.483,E2 14302.483} C_VEL
LIN {X 0,Y 320.918,Z 1074.699,A -85,B 0,C 180,E1 14299.407,E2 14299.407} C_VEL
LIN {X 0,Y 321.172,Z 1067.741,A -85,B 0,C 180,E1 14296.24,E2 14296.24} C_VEL
LIN {X 0,Y 321.936,Z 1059.208,A -85,B 0,C 180,E1 14293.211,E2 14293.211} C_VEL
LIN {X 0,Y 323.24,Z 1049.001,A -85,B 0,C 180,E1 14290.295,E2 14290.295} C_VEL
LIN {X 0,Y 325.058,Z 1037.365,A -85,B 0,C 180,E1 14287.578,E2 14287.578} C_VEL
LIN {X 0,Y 327.388,Z 1023.777,A -85,B 0,C 180,E1 14284.976,E2 14284.976} C_VEL
LIN {X 0,Y 329.963,Z 1009.266,A -85,B 0,C 180,E1 14282.705,E2 14282.705} C_VEL
LIN {X 0,Y 332.601,Z 994.142,A -85,B 0,C 180,E1 14280.762,E2 14280.762} C_VEL
LIN {X 0,Y 335.304,Z 977.579,A -85,B 0,C 180,E1 14279.043,E2 14279.043} C_VEL
LIN {X 0,Y 337.873,Z 960.174,A -85,B 0,C 180,E1 14277.613,E2 14277.613} C_VEL
LIN {X 0,Y 340.099,Z 942.503,A -85,B 0,C 180,E1 14276.497,E2 14276.497} C_VEL
LIN {X 0,Y 342.004,Z 923.501,A -85,B 0,C 180,E1 14275.632,E2 14275.632} C_VEL
LIN {X 0,Y 343.15,Z 903.846,A -85,B 0,C 180,E1 14275.042,E2 14275.042} C_VEL
LIN {X 0,Y 347.745,Z 746.591,A -85,B 0,C 180,E1 14271.802,E2 14271.802} C_VEL
LIN {X 0,Y 343.51,Z 705.777,A -85,B 0,C 180,E1 14270.371,E2 14270.371} C_VEL
LIN {X 0,Y 344.705,Z 697.431,A -85,B 0,C 180,E1 14269.333,E2 14269.333} C_VEL
LIN {X 0,Y 338.246,Z 677.255,A -85,B 0,C 180,E1 14265.672,E2 14265.672} C_VEL
LIN {X 0,Y 332.196,Z 659.958,A -85,B 0,C 180,E1 14262.159,E2 14262.159} C_VEL
LIN {X 0,Y 326.909,Z 646.165,A -85,B 0,C 180,E1 14259.003,E2 14259.003} C_VEL
LIN {X 0,Y 327.412,Z 642.128,A -85,B 0,C 180,E1 14257.15,E2 14257.15} C_VEL
LIN {X 0,Y 327.326,Z 642.163,A -85,B 0,C 180,E1 14254.744,E2 14254.744} C_VEL
LIN {X 0,Y 328.752,Z 644.836,A -85,B 0,C 180,E1 14250.727,E2 14250.727} C_VEL
LIN {X 0,Y 330.484,Z 646.66,A -85,B 0,C 180,E1 14248.753,E2 14248.753} C_VEL
LIN {X 0,Y 332.098,Z 650.175,A -85,B 0,C 180,E1 14246.847,E2 14246.847} C_VEL
LIN {X 0,Y 333.364,Z 651.919,A -85,B 0,C 180,E1 14245.779,E2 14245.779} C_VEL
LIN {X 0,Y 335.296,Z 655.716,A -85,B 0,C 180,E1 14244.113,E2 14244.113} C_VEL
LIN {X 0,Y 337.913,Z 661.263,A -85,B 0,C 180,E1 14242.072,E2 14242.072} C_VEL
LIN {X 0,Y 340.942,Z 668.308,A -85,B 0,C 180,E1 14239.888,E2 14239.888} C_VEL
LIN {X 0,Y 344.042,Z 676.977,A -85,B 0,C 180,E1 14237.589,E2 14237.589} C_VEL
LIN {X 0,Y 347.075,Z 687.839,A -85,B 0,C 180,E1 14235.186,E2 14235.186} C_VEL
LIN {X 0,Y 348.719,Z 696.69,A -85,B 0,C 180,E1 14233.514,E2 14233.514} C_VEL
LIN {X 0,Y 345.991,Z 730.633,A -85,B 0,C 180,E1 14228.977,E2 14228.977} C_VEL
LIN {X 0,Y 345.751,Z 736.271,A -85,B 0,C 180,E1 14228.272,E2 14228.272} C_VEL
LIN {X 0,Y 345.953,Z 739.246,A -85,B 0,C 180,E1 14228.125,E2 14228.125} C_VEL
LIN {X 0,Y 339.469,Z 855.778,A -85,B 0,C 180,E1 14224.857,E2 14224.857} C_VEL
LIN {X 0,Y 338.962,Z 878.374,A -85,B 0,C 180,E1 14224.086,E2 14224.086} C_VEL
LIN {X 0,Y 338.167,Z 894.574,A -85,B 0,C 180,E1 14223.22,E2 14223.22} C_VEL
LIN {X 0,Y 336.874,Z 910.292,A -85,B 0,C 180,E1 14222.041,E2 14222.041} C_VEL
LIN {X 0,Y 335.358,Z 924.185,A -85,B 0,C 180,E1 14220.683,E2 14220.683} C_VEL
LIN {X 0,Y 333.479,Z 937.768,A -85,B 0,C 180,E1 14218.969,E2 14218.969} C_VEL
LIN {X 0,Y 331.687,Z 948.749,A -85,B 0,C 180,E1 14217.235,E2 14217.235} C_VEL
LIN {X 0,Y 329.553,Z 960.171,A -85,B 0,C 180,E1 14214.952,E2 14214.952} C_VEL
LIN {X 0,Y 327.831,Z 968.592,A -85,B 0,C 180,E1 14212.816,E2 14212.816} C_VEL
LIN {X 0,Y 326.128,Z 976.24,A -85,B 0,C 180,E1 14210.292,E2 14210.292} C_VEL
LIN {X 0,Y 324.78,Z 981.989,A -85,B 0,C 180,E1 14207.735,E2 14207.735} C_VEL
LIN {X 0,Y 323.677,Z 986.213,A -85,B 0,C 180,E1 14204.96,E2 14204.96} C_VEL
LIN {X 0,Y 322.93,Z 988.619,A -85,B 0,C 180,E1 14202.15,E2 14202.15} C_VEL
LIN {X 0,Y 322.485,Z 989.183,A -85,B 0,C 180,E1 14199.301,E2 14199.301} C_VEL
LIN {X 0,Y 322.317,Z 988.087,A -85,B 0,C 180,E1 14196.604,E2 14196.604} C_VEL
LIN {X 0,Y 322.387,Z 985.002,A -85,B 0,C 180,E1 14193.679,E2 14193.679} C_VEL
LIN {X 0,Y 322.741,Z 980.22,A -85,B 0,C 180,E1 14190.886,E2 14190.886} C_VEL
LIN {X 0,Y 323.408,Z 973.341,A -85,B 0,C 180,E1 14188.084,E2 14188.084} C_VEL
LIN {X 0,Y 324.266,Z 965.438,A -85,B 0,C 180,E1 14185.648,E2 14185.648} C_VEL
LIN {X 0,Y 325.477,Z 954.973,A -85,B 0,C 180,E1 14183.126,E2 14183.126} C_VEL
LIN {X 0,Y 326.797,Z 943.362,A -85,B 0,C 180,E1 14180.929,E2 14180.929} C_VEL
LIN {X 0,Y 328.124,Z 931.162,A -85,B 0,C 180,E1 14179.069,E2 14179.069} C_VEL
LIN {X 0,Y 329.486,Z 916.701,A -85,B 0,C 180,E1 14177.322,E2 14177.322} C_VEL
LIN {X 0,Y 330.659,Z 902.042,A -85,B 0,C 180,E1 14175.934,E2 14175.934} C_VEL
LIN {X 0,Y 331.671,Z 885.386,A -85,B 0,C 180,E1 14174.745,E2 14174.745} C_VEL
LIN {X 0,Y 332.3,Z 868.518,A -85,B 0,C 180,E1 14173.906,E2 14173.906} C_VEL
LIN {X 0,Y 332.605,Z 848.946,A -85,B 0,C 180,E1 14173.303,E2 14173.303} C_VEL
LIN {X 0,Y 336.436,Z 729.541,A -85,B 0,C 180,E1 14170.278,E2 14170.278} C_VEL
LIN {X 0,Y 335.087,Z 720.752,A -85,B 0,C 180,E1 14169.907,E2 14169.907} C_VEL
LIN {X 0,Y 336.774,Z 687.458,A -85,B 0,C 180,E1 14165.481,E2 14165.481} C_VEL
LIN {X 0,Y 336.844,Z 682.122,A -85,B 0,C 180,E1 14164.745,E2 14164.745} C_VEL
LIN {X 0,Y 331.823,Z 663.364,A -85,B 0,C 180,E1 14161.622,E2 14161.622} C_VEL
LIN {X 0,Y 325.873,Z 645.036,A -85,B 0,C 180,E1 14158.398,E2 14158.398} C_VEL
LIN {X 0,Y 324.525,Z 641.008,A -85,B 0,C 180,E1 14157.576,E2 14157.576} C_VEL
LIN {X 0,Y 324.547,Z 641.257,A -85,B 0,C 180,E1 14157.326,E2 14157.326} C_VEL
LIN {X 0,Y 328.657,Z 653.431,A -85,B 0,C 180,E1 14153.963,E2 14153.963} C_VEL
LIN {X 0,Y 332.883,Z 667.726,A -85,B 0,C 180,E1 14150.391,E2 14150.391} C_VEL
LIN {X 0,Y 336.63,Z 682.574,A -85,B 0,C 180,E1 14146.923,E2 14146.923} C_VEL
LIN {X 0,Y 337.659,Z 687.633,A -85,B 0,C 180,E1 14145.809,E2 14145.809} C_VEL
LIN {X 0,Y 336.427,Z 696.095,A -85,B 0,C 180,E1 14144.332,E2 14144.332} C_VEL
LIN {X 0,Y 337.861,Z 704.08,A -85,B 0,C 180,E1 14143.93,E2 14143.93} C_VEL
LIN {X 0,Y 343.491,Z 735.391,A -85,B 0,C 180,E1 14142.627,E2 14142.627} C_VEL
LIN {X 0,Y 339.921,Z 852.535,A -85,B 0,C 180,E1 14140.112,E2 14140.112} C_VEL
LIN {X 0,Y 339.183,Z 868.214,A -85,B 0,C 180,E1 14139.508,E2 14139.508} C_VEL
LIN {X 0,Y 337.705,Z 875.748,A -85,B 0,C 180,E1 14139.209,E2 14139.209} C_VEL
LIN {X 0,Y 331.844,Z 891.128,A -85,B 0,C 180,E1 14138.612,E2 14138.612} C_VEL
LIN {X 0,Y 329.392,Z 899.042,A -85,B 0,C 180,E1 14138.115,E2 14138.115} C_VEL
LIN {X 0,Y 329.085,Z 900.968,A -85,B 0,C 180,E1 14137.955,E2 14137.955} C_VEL
LIN {X 0,Y 327.154,Z 915.479,A -85,B 0,C 180,E1 14136.493,E2 14136.493} C_VEL
LIN {X 0,Y 324.931,Z 929.624,A -85,B 0,C 180,E1 14134.678,E2 14134.678} C_VEL
LIN {X 0,Y 322.696,Z 942.459,A -85,B 0,C 180,E1 14132.618,E2 14132.618} C_VEL
LIN {X 0,Y 320.568,Z 953.736,A -85,B 0,C 180,E1 14130.358,E2 14130.358} C_VEL
LIN {X 0,Y 318.6,Z 963.721,A -85,B 0,C 180,E1 14127.842,E2 14127.842} C_VEL
LIN {X 0,Y 316.952,Z 972.256,A -85,B 0,C 180,E1 14125.114,E2 14125.114} C_VEL
LIN {X 0,Y 315.743,Z 978.87,A -85,B 0,C 180,E1 14122.357,E2 14122.357} C_VEL
LIN {X 0,Y 314.902,Z 984.037,A -85,B 0,C 180,E1 14119.388,E2 14119.388} C_VEL
LIN {X 0,Y 314.436,Z 987.683,A -85,B 0,C 180,E1 14116.203,E2 14116.203} C_VEL
LIN {X 0,Y 314.362,Z 989.442,A -85,B 0,C 180,E1 14113.176,E2 14113.176} C_VEL
LIN {X 0,Y 314.662,Z 989.499,A -85,B 0,C 180,E1 14109.93,E2 14109.93} C_VEL
LIN {X 0,Y 315.43,Z 987.738,A -85,B 0,C 180,E1 14106.658,E2 14106.658} C_VEL
LIN {X 0,Y 316.647,Z 984.241,A -85,B 0,C 180,E1 14103.563,E2 14103.563} C_VEL
LIN {X 0,Y 318.439,Z 978.773,A -85,B 0,C 180,E1 14100.465,E2 14100.465} C_VEL
LIN {X 0,Y 320.729,Z 971.694,A -85,B 0,C 180,E1 14097.575,E2 14097.575} C_VEL
LIN {X 0,Y 323.406,Z 962.957,A -85,B 0,C 180,E1 14094.898,E2 14094.898} C_VEL
LIN {X 0,Y 326.369,Z 952.696,A -85,B 0,C 180,E1 14092.436,E2 14092.436} C_VEL
LIN {X 0,Y 329.512,Z 940.9,A -85,B 0,C 180,E1 14090.19,E2 14090.19} C_VEL
LIN {X 0,Y 332.627,Z 927.621,A -85,B 0,C 180,E1 14088.201,E2 14088.201} C_VEL
LIN {X 0,Y 335.534,Z 913.301,A -85,B 0,C 180,E1 14086.5,E2 14086.5} C_VEL
LIN {X 0,Y 338.027,Z 898.599,A -85,B 0,C 180,E1 14085.133,E2 14085.133} C_VEL
LIN {X 0,Y 340.13,Z 882.318,A -85,B 0,C 180,E1 14083.989,E2 14083.989} C_VEL
LIN {X 0,Y 341.661,Z 865.204,A -85,B 0,C 180,E1 14083.124,E2 14083.124} C_VEL
LIN {X 0,Y 342.5,Z 847.871,A -85,B 0,C 180,E1 14082.564,E2 14082.564} C_VEL
LIN {X 0,Y 346.96,Z 738.952,A -85,B 0,C 180,E1 14080.164,E2 14080.164} C_VEL
LIN {X 0,Y 341.188,Z 711.231,A -85,B 0,C 180,E1 14078.498,E2 14078.498} C_VEL
LIN {X 0,Y 338.945,Z 702.372,A -85,B 0,C 180,E1 14077.876,E2 14077.876} C_VEL
LIN {X 0,Y 336.538,Z 697.847,A -85,B 0,C 180,E1 14077.308,E2 14077.308} C_VEL
LIN {X 0,Y 335.549,Z 694.045,A -85,B 0,C 180,E1 14076.369,E2 14076.369} C_VEL
LIN {X 0,Y 332.502,Z 682.359,A -85,B 0,C 180,E1 14072.969,E2 14072.969} C_VEL
LIN {X 0,Y 329.164,Z 671.655,A -85,B 0,C 180,E1 14069.478,E2 14069.478} C_VEL
LIN {X 0,Y 325.641,Z 661.901,A -85,B 0,C 180,E1 14065.849,E2 14065.849} C_VEL
LIN {X 0,Y 322.804,Z 654.748,A -85,B 0,C 180,E1 14062.779,E2 14062.779} C_VEL
LIN {X 0,Y 320.97,Z 650.515,A -85,B 0,C 180,E1 14060.801,E2 14060.801} C_VEL
LIN {X 0,Y 319.573,Z 647.266,A -85,B 0,C 180,E1 14059.179,E2 14059.179} C_VEL
LIN {X 0,Y 317.836,Z 643.345,A -85,B 0,C 180,E1 14057.012,E2 14057.012} C_VEL
LIN {X 0,Y 315.905,Z 639.141,A -85,B 0,C 180,E1 14054.418,E2 14054.418} C_VEL
LIN {X 0,Y 314.177,Z 635.178,A -85,B 0,C 180,E1 14051.423,E2 14051.423} C_VEL
LIN {X 0,Y 314.161,Z 635.086,A -85,B 0,C 180,E1 14046.947,E2 14046.947} C_VEL
LIN {X 0,Y 314.164,Z 635.089,A -85,B 0,C 180,E1 14042.372,E2 14042.372} C_VEL
LIN {X 0,Y 314.168,Z 635.099,A -85,B 0,C 180,E1 14037.994,E2 14037.994} C_VEL
LIN {X 0,Y 314.175,Z 635.097,A -85,B 0,C 180,E1 14033.422,E2 14033.422} C_VEL
LIN {X 0,Y 314.171,Z 635.088,A -85,B 0,C 180,E1 14028.992,E2 14028.992} C_VEL
LIN {X 0,Y 314.17,Z 635.084,A -85,B 0,C 180,E1 14024.495,E2 14024.495} C_VEL
LIN {X 0,Y 314.165,Z 635.082,A -85,B 0,C 180,E1 14020.091,E2 14020.091} C_VEL
LIN {X 0,Y 314.207,Z 635.419,A -85,B 0,C 180,E1 14017.453,E2 14017.453} C_VEL
LIN {X 0,Y 316.156,Z 639.463,A -85,B 0,C 180,E1 14014.727,E2 14014.727} C_VEL
LIN {X 0,Y 317.049,Z 641.434,A -85,B 0,C 180,E1 14013.599,E2 14013.599} C_VEL
LIN {X 0,Y 319.268,Z 645.589,A -85,B 0,C 180,E1 14011.268,E2 14011.268} C_VEL
LIN {X 0,Y 321.654,Z 650.524,A -85,B 0,C 180,E1 14008.935,E2 14008.935} C_VEL
LIN {X 0,Y 323.908,Z 655.339,A -85,B 0,C 180,E1 14006.882,E2 14006.882} C_VEL
LIN {X 0,Y 327.039,Z 662.025,A -85,B 0,C 180,E1 14004.272,E2 14004.272} C_VEL
LIN {X 0,Y 331.618,Z 672.815,A -85,B 0,C 180,E1 14000.716,E2 14000.716} C_VEL
LIN {X 0,Y 336.374,Z 685.246,A -85,B 0,C 180,E1 13997.239,E2 13997.239} C_VEL
LIN {X 0,Y 340.756,Z 698.547,A -85,B 0,C 180,E1 13994.038,E2 13994.038} C_VEL
LIN {X 0,Y 343.029,Z 706.165,A -85,B 0,C 180,E1 13992.455,E2 13992.455} C_VEL
LIN {X 0,Y 343.685,Z 708.454,A -85,B 0,C 180,E1 13992.282,E2 13992.282} C_VEL
LIN {X 0,Y 347.229,Z 740.433,A -85,B 0,C 180,E1 13990.843,E2 13990.843} C_VEL
LIN {X 0,Y 347.958,Z 752.254,A -85,B 0,C 180,E1 13990.412,E2 13990.412} C_VEL
LIN {X 0,Y 341.626,Z 908.43,A -85,B 0,C 180,E1 13987.051,E2 13987.051} C_VEL
LIN {X 0,Y 339.866,Z 927.391,A -85,B 0,C 180,E1 13986.381,E2 13986.381} C_VEL
LIN {X 0,Y 337.489,Z 944.86,A -85,B 0,C 180,E1 13985.498,E2 13985.498} C_VEL
LIN {X 0,Y 334.556,Z 962.491,A -85,B 0,C 180,E1 13984.288,E2 13984.288} C_VEL
LIN {X 0,Y 331.32,Z 979.264,A -85,B 0,C 180,E1 13982.799,E2 13982.799} C_VEL
LIN {X 0,Y 327.934,Z 995.227,A -85,B 0,C 180,E1 13981.015,E2 13981.015} C_VEL
LIN {X 0,Y 324.385,Z 1010.905,A -85,B 0,C 180,E1 13978.841,E2 13978.841} C_VEL
LIN {X 0,Y 321.138,Z 1025.012,A -85,B 0,C 180,E1 13976.438,E2 13976.438} C_VEL
LIN {X 0,Y 318.226,Z 1038.106,A -85,B 0,C 180,E1 13973.714,E2 13973.714} C_VEL
LIN {X 0,Y 315.866,Z 1049.691,A -85,B 0,C 180,E1 13970.764,E2 13970.764} C_VEL
LIN {X 0,Y 314.165,Z 1059.783,A -85,B 0,C 180,E1 13967.598,E2 13967.598} C_VEL
LIN {X 0,Y 313.155,Z 1068.342,A -85,B 0,C 180,E1 13964.232,E2 13964.232} C_VEL
LIN {X 0,Y 312.833,Z 1074.92,A -85,B 0,C 180,E1 13960.869,E2 13960.869} C_VEL
LIN {X 0,Y 312.962,Z 1079.646,A -85,B 0,C 180,E1 13957.526,E2 13957.526} C_VEL
LIN {X 0,Y 313.292,Z 1082.464,A -85,B 0,C 180,E1 13954.392,E2 13954.392} C_VEL
LIN {X 0,Y 313.558,Z 1083.725,A -85,B 0,C 180,E1 13951.279,E2 13951.279} C_VEL
LIN {X 0,Y 313.568,Z 1083.467,A -85,B 0,C 180,E1 13948.355,E2 13948.355} C_VEL
LIN {X 0,Y 313.343,Z 1081.803,A -85,B 0,C 180,E1 13945.424,E2 13945.424} C_VEL
LIN {X 0,Y 313.059,Z 1078.413,A -85,B 0,C 180,E1 13942.291,E2 13942.291} C_VEL
LIN {X 0,Y 312.965,Z 1072.982,A -85,B 0,C 180,E1 13938.948,E2 13938.948} C_VEL
LIN {X 0,Y 313.308,Z 1065.529,A -85,B 0,C 180,E1 13935.586,E2 13935.586} C_VEL
LIN {X 0,Y 314.225,Z 1056.459,A -85,B 0,C 180,E1 13932.404,E2 13932.404} C_VEL
LIN {X 0,Y 315.716,Z 1045.862,A -85,B 0,C 180,E1 13929.418,E2 13929.418} C_VEL
LIN {X 0,Y 317.736,Z 1033.784,A -85,B 0,C 180,E1 13926.64,E2 13926.64} C_VEL
LIN {X 0,Y 320.214,Z 1020.082,A -85,B 0,C 180,E1 13924.062,E2 13924.062} C_VEL
LIN {X 0,Y 323.021,Z 1004.912,A -85,B 0,C 180,E1 13921.732,E2 13921.732} C_VEL
LIN {X 0,Y 325.818,Z 989.296,A -85,B 0,C 180,E1 13919.782,E2 13919.782} C_VEL
LIN {X 0,Y 328.632,Z 972.407,A -85,B 0,C 180,E1 13918.087,E2 13918.087} C_VEL
LIN {X 0,Y 331.272,Z 954.513,A -85,B 0,C 180,E1 13916.679,E2 13916.679} C_VEL
LIN {X 0,Y 333.5,Z 936.588,A -85,B 0,C 180,E1 13915.617,E2 13915.617} C_VEL
LIN {X 0,Y 335.297,Z 917.348,A -85,B 0,C 180,E1 13914.813,E2 13914.813} C_VEL
LIN {X 0,Y 336.249,Z 896.944,A -85,B 0,C 180,E1 13914.277,E2 13914.277} C_VEL
LIN {X 0,Y 340.792,Z 747.555,A -85,B 0,C 180,E1 13911.157,E2 13911.157} C_VEL
LIN {X 0,Y 336.524,Z 705.785,A -85,B 0,C 180,E1 13909.665,E2 13909.665} C_VEL
LIN {X 0,Y 337.408,Z 700.148,A -85,B 0,C 180,E1 13908.966,E2 13908.966} C_VEL
LIN {X 0,Y 331.064,Z 680.09,A -85,B 0,C 180,E1 13905.213,E2 13905.213} C_VEL
LIN {X 0,Y 325.044,Z 662.858,A -85,B 0,C 180,E1 13901.626,E2 13901.626} C_VEL
LIN {X 0,Y 323.619,Z 658.83,A -85,B 0,C 180,E1 13900.685,E2 13900.685} C_VEL
LIN {X 0,Y 323.754,Z 653.266,A -85,B 0,C 180,E1 13898.597,E2 13898.597} C_VEL
LIN {X 0,Y 324.419,Z 649.506,A -85,B 0,C 180,E1 13896.94,E2 13896.94} C_VEL
LIN {X 0,Y 324.251,Z 649.55,A -85,B 0,C 180,E1 13894.782,E2 13894.782} C_VEL
LIN {X 0,Y 325.387,Z 652.05,A -85,B 0,C 180,E1 13890.874,E2 13890.874} C_VEL
LIN {X 0,Y 326.772,Z 653.449,A -85,B 0,C 180,E1 13889.111,E2 13889.111} C_VEL
LIN {X 0,Y 328.285,Z 657.163,A -85,B 0,C 180,E1 13886.988,E2 13886.988} C_VEL
LIN {X 0,Y 329.335,Z 658.78,A -85,B 0,C 180,E1 13886.017,E2 13886.017} C_VEL
LIN {X 0,Y 331.642,Z 663.786,A -85,B 0,C 180,E1 13883.828,E2 13883.828} C_VEL
LIN {X 0,Y 334.494,Z 670.17,A -85,B 0,C 180,E1 13881.48,E2 13881.48} C_VEL
LIN {X 0,Y 337.996,Z 679.576,A -85,B 0,C 180,E1 13878.803,E2 13878.803} C_VEL
LIN {X 0,Y 340.699,Z 689.667,A -85,B 0,C 180,E1 13876.329,E2 13876.329} C_VEL
LIN {X 0,Y 342.843,Z 700.043,A -85,B 0,C 180,E1 13874.223,E2 13874.223} C_VEL
LIN {X 0,Y 339.748,Z 734.303,A -85,B 0,C 180,E1 13869.571,E2 13869.571} C_VEL
LIN {X 0,Y 339.66,Z 737.888,A -85,B 0,C 180,E1 13869.136,E2 13869.136} C_VEL
LIN {X 0,Y 339.91,Z 740.862,A -85,B 0,C 180,E1 13868.979,E2 13868.979} C_VEL
LIN {X 0,Y 332.934,Z 857.229,A -85,B 0,C 180,E1 13865.617,E2 13865.617} C_VEL
LIN {X 0,Y 332.314,Z 880.107,A -85,B 0,C 180,E1 13864.8,E2 13864.8} C_VEL
LIN {X 0,Y 331.437,Z 896.627,A -85,B 0,C 180,E1 13863.892,E2 13863.892} C_VEL
LIN {X 0,Y 330.056,Z 912.159,A -85,B 0,C 180,E1 13862.691,E2 13862.691} C_VEL
LIN {X 0,Y 328.424,Z 925.868,A -85,B 0,C 180,E1 13861.308,E2 13861.308} C_VEL
LIN {X 0,Y 326.32,Z 939.96,A -85,B 0,C 180,E1 13859.473,E2 13859.473} C_VEL
LIN {X 0,Y 324.23,Z 951.737,A -85,B 0,C 180,E1 13857.525,E2 13857.525} C_VEL
LIN {X 0,Y 322.059,Z 962.551,A -85,B 0,C 180,E1 13855.261,E2 13855.261} C_VEL
LIN {X 0,Y 320.024,Z 971.526,A -85,B 0,C 180,E1 13852.82,E2 13852.82} C_VEL
LIN {X 0,Y 318.277,Z 978.839,A -85,B 0,C 180,E1 13850.233,E2 13850.233} C_VEL
LIN {X 0,Y 316.791,Z 984.524,A -85,B 0,C 180,E1 13847.421,E2 13847.421} C_VEL
LIN {X 0,Y 315.75,Z 988.106,A -85,B 0,C 180,E1 13844.762,E2 13844.762} C_VEL
LIN {X 0,Y 314.983,Z 990.125,A -85,B 0,C 180,E1 13841.875,E2 13841.875} C_VEL
LIN {X 0,Y 314.549,Z 990.392,A -85,B 0,C 180,E1 13838.949,E2 13838.949} C_VEL
LIN {X 0,Y 314.39,Z 988.746,A -85,B 0,C 180,E1 13835.978,E2 13835.978} C_VEL
LIN {X 0,Y 314.51,Z 985.481,A -85,B 0,C 180,E1 13833.164,E2 13833.164} C_VEL
LIN {X 0,Y 314.922,Z 980.282,A -85,B 0,C 180,E1 13830.311,E2 13830.311} C_VEL
LIN {X 0,Y 315.616,Z 973.537,A -85,B 0,C 180,E1 13827.629,E2 13827.629} C_VEL
LIN {X 0,Y 316.666,Z 964.326,A -85,B 0,C 180,E1 13824.864,E2 13824.864} C_VEL
LIN {X 0,Y 317.812,Z 954.744,A -85,B 0,C 180,E1 13822.613,E2 13822.613} C_VEL
LIN {X 0,Y 319.192,Z 943.063,A -85,B 0,C 180,E1 13820.408,E2 13820.408} C_VEL
LIN {X 0,Y 320.619,Z 930.073,A -85,B 0,C 180,E1 13818.457,E2 13818.457} C_VEL
LIN {X 0,Y 321.958,Z 916.236,A -85,B 0,C 180,E1 13816.794,E2 13816.794} C_VEL
LIN {X 0,Y 323.184,Z 900.887,A -85,B 0,C 180,E1 13815.363,E2 13815.363} C_VEL
LIN {X 0,Y 324.155,Z 884.983,A -85,B 0,C 180,E1 13814.243,E2 13814.243} C_VEL
LIN {X 0,Y 324.815,Z 867.073,A -85,B 0,C 180,E1 13813.369,E2 13813.369} C_VEL
LIN {X 0,Y 325.532,Z 830.82,A -85,B 0,C 180,E1 13812.351,E2 13812.351} C_VEL
LIN {X 0,Y 329.077,Z 730.52,A -85,B 0,C 180,E1 13809.74,E2 13809.74} C_VEL
LIN {X 0,Y 327.758,Z 721.444,A -85,B 0,C 180,E1 13809.329,E2 13809.329} C_VEL
LIN {X 0,Y 329.519,Z 688.438,A -85,B 0,C 180,E1 13804.899,E2 13804.899} C_VEL
LIN {X 0,Y 329.514,Z 684.6,A -85,B 0,C 180,E1 13804.36,E2 13804.36} C_VEL
LIN {X 0,Y 324.616,Z 666.289,A -85,B 0,C 180,E1 13801.266,E2 13801.266} C_VEL
LIN {X 0,Y 318.812,Z 648.385,A -85,B 0,C 180,E1 13798.063,E2 13798.063} C_VEL
LIN {X 0,Y 318.05,Z 645.967,A -85,B 0,C 180,E1 13797.525,E2 13797.525} C_VEL
LIN {X 0,Y 318.106,Z 646.473,A -85,B 0,C 180,E1 13797.187,E2 13797.187} C_VEL
LIN {X 0,Y 322,Z 658.247,A -85,B 0,C 180,E1 13793.906,E2 13793.906} C_VEL
LIN {X 0,Y 326.019,Z 672.144,A -85,B 0,C 180,E1 13790.371,E2 13790.371} C_VEL
LIN {X 0,Y 329.612,Z 686.69,A -85,B 0,C 180,E1 13786.931,E2 13786.931} C_VEL
LIN {X 0,Y 330.278,Z 690.064,A -85,B 0,C 180,E1 13786.172,E2 13786.172} C_VEL
LIN {X 0,Y 329.335,Z 696.687,A -85,B 0,C 180,E1 13785.03,E2 13785.03} C_VEL
LIN {X 0,Y 336.53,Z 736.491,A -85,B 0,C 180,E1 13783.28,E2 13783.28} C_VEL
LIN {X 0,Y 332.818,Z 853.197,A -85,B 0,C 180,E1 13780.73,E2 13780.73} C_VEL
LIN {X 0,Y 331.938,Z 870.495,A -85,B 0,C 180,E1 13780.035,E2 13780.035} C_VEL
LIN {X 0,Y 330.593,Z 887.128,A -85,B 0,C 180,E1 13779.049,E2 13779.049} C_VEL
LIN {X 0,Y 329.085,Z 900.968,A -85,B 0,C 180,E1 13777.955,E2 13777.955} C_VEL
LIN {X 0,Y 327.348,Z 907.84,A -85,B 0,C 180,E1 13777.398,E2 13777.398} C_VEL
LIN {X 0,Y 320.676,Z 921.777,A -85,B 0,C 180,E1 13776.24,E2 13776.24} C_VEL
LIN {X 0,Y 317.882,Z 928.891,A -85,B 0,C 180,E1 13775.422,E2 13775.422} C_VEL
LIN {X 0,Y 317.503,Z 930.59,A -85,B 0,C 180,E1 13775.179,E2 13775.179} C_VEL
LIN {X 0,Y 315.19,Z 943.333,A -85,B 0,C 180,E1 13773.092,E2 13773.092} C_VEL
LIN {X 0,Y 312.923,Z 954.856,A -85,B 0,C 180,E1 13770.733,E2 13770.733} C_VEL
LIN {X 0,Y 310.87,Z 964.838,A -85,B 0,C 180,E1 13768.157,E2 13768.157} C_VEL
LIN {X 0,Y 309.148,Z 973.378,A -85,B 0,C 180,E1 13765.363,E2 13765.363} C_VEL
LIN {X 0,Y 307.884,Z 980.001,A -85,B 0,C 180,E1 13762.537,E2 13762.537} C_VEL
LIN {X 0,Y 307.004,Z 985.181,A -85,B 0,C 180,E1 13759.492,E2 13759.492} C_VEL
LIN {X 0,Y 306.52,Z 988.844,A -85,B 0,C 180,E1 13756.225,E2 13756.225} C_VEL
LIN {X 0,Y 306.451,Z 990.63,A -85,B 0,C 180,E1 13753.12,E2 13753.12} C_VEL
LIN {X 0,Y 306.779,Z 990.716,A -85,B 0,C 180,E1 13749.79,E2 13749.79} C_VEL
LIN {X 0,Y 307.602,Z 988.987,A -85,B 0,C 180,E1 13746.434,E2 13746.434} C_VEL
LIN {X 0,Y 308.902,Z 985.542,A -85,B 0,C 180,E1 13743.262,E2 13743.262} C_VEL
LIN {X 0,Y 310.806,Z 980.118,A -85,B 0,C 180,E1 13740.091,E2 13740.091} C_VEL
LIN {X 0,Y 313.284,Z 972.938,A -85,B 0,C 180,E1 13737.075,E2 13737.075} C_VEL
LIN {X 0,Y 316.059,Z 964.437,A -85,B 0,C 180,E1 13734.393,E2 13734.393} C_VEL
LIN {X 0,Y 319.248,Z 954,A -85,B 0,C 180,E1 13731.824,E2 13731.824} C_VEL
LIN {X 0,Y 322.595,Z 942.099,A -85,B 0,C 180,E1 13729.509,E2 13729.509} C_VEL
LIN {X 0,Y 325.789,Z 929.196,A -85,B 0,C 180,E1 13727.532,E2 13727.532} C_VEL
LIN {X 0,Y 328.864,Z 914.817,A -85,B 0,C 180,E1 13725.784,E2 13725.784} C_VEL
LIN {X 0,Y 331.516,Z 900.004,A -85,B 0,C 180,E1 13724.374,E2 13724.374} C_VEL
LIN {X 0,Y 333.722,Z 883.958,A -85,B 0,C 180,E1 13723.215,E2 13723.215} C_VEL
LIN {X 0,Y 335.384,Z 866.512,A -85,B 0,C 180,E1 13722.309,E2 13722.309} C_VEL
LIN {X 0,Y 336.298,Z 849.161,A -85,B 0,C 180,E1 13721.729,E2 13721.729} C_VEL
LIN {X 0,Y 340.972,Z 740.58,A -85,B 0,C 180,E1 13719.301,E2 13719.301} C_VEL
LIN {X 0,Y 335.247,Z 712.512,A -85,B 0,C 180,E1 13717.557,E2 13717.557} C_VEL
LIN {X 0,Y 333.779,Z 706.82,A -85,B 0,C 180,E1 13717.129,E2 13717.129} C_VEL
LIN {X 0,Y 328.754,Z 697.504,A -85,B 0,C 180,E1 13715.89,E2 13715.89} C_VEL
LIN {X 0,Y 325.745,Z 685.884,A -85,B 0,C 180,E1 13712.425,E2 13712.425} C_VEL
LIN {X 0,Y 322.334,Z 674.968,A -85,B 0,C 180,E1 13708.738,E2 13708.738} C_VEL
LIN {X 0,Y 319.281,Z 666.356,A -85,B 0,C 180,E1 13705.406,E2 13705.406} C_VEL
LIN {X 0,Y 316.695,Z 659.671,A -85,B 0,C 180,E1 13702.459,E2 13702.459} C_VEL
LIN {X 0,Y 314.088,Z 653.221,A -85,B 0,C 180,E1 13699.334,E2 13699.334} C_VEL
LIN {X 0,Y 312.043,Z 648.763,A -85,B 0,C 180,E1 13696.761,E2 13696.761} C_VEL
LIN {X 0,Y 310.195,Z 644.682,A -85,B 0,C 180,E1 13694.181,E2 13694.181} C_VEL
LIN {X 0,Y 308.062,Z 640.267,A -85,B 0,C 180,E1 13690.851,E2 13690.851} C_VEL
LIN {X 0,Y 306.235,Z 636.158,A -85,B 0,C 180,E1 13686.751,E2 13686.751} C_VEL
LIN {X 0,Y 306.227,Z 636.074,A -85,B 0,C 180,E1 13682.246,E2 13682.246} C_VEL
LIN {X 0,Y 306.232,Z 636.08,A -85,B 0,C 180,E1 13677.755,E2 13677.755} C_VEL
LIN {X 0,Y 306.238,Z 636.087,A -85,B 0,C 180,E1 13673.25,E2 13673.25} C_VEL
LIN {X 0,Y 306.23,Z 636.082,A -85,B 0,C 180,E1 13668.703,E2 13668.703} C_VEL
LIN {X 0,Y 306.225,Z 636.077,A -85,B 0,C 180,E1 13664.276,E2 13664.276} C_VEL
LIN {X 0,Y 306.288,Z 636.507,A -85,B 0,C 180,E1 13661.934,E2 13661.934} C_VEL
LIN {X 0,Y 308.976,Z 641.748,A -85,B 0,C 180,E1 13657.351,E2 13657.351} C_VEL
LIN {X 0,Y 311.473,Z 646.633,A -85,B 0,C 180,E1 13654.115,E2 13654.115} C_VEL
LIN {X 0,Y 313.813,Z 651.387,A -85,B 0,C 180,E1 13651.45,E2 13651.45} C_VEL
LIN {X 0,Y 316.073,Z 656.106,A -85,B 0,C 180,E1 13649.172,E2 13649.172} C_VEL
LIN {X 0,Y 318.509,Z 661.421,A -85,B 0,C 180,E1 13646.892,E2 13646.892} C_VEL
LIN {X 0,Y 321.554,Z 668.224,A -85,B 0,C 180,E1 13644.227,E2 13644.227} C_VEL
LIN {X 0,Y 325.614,Z 677.897,A -85,B 0,C 180,E1 13640.975,E2 13640.975} C_VEL
LIN {X 0,Y 330.151,Z 690.003,A -85,B 0,C 180,E1 13637.519,E2 13637.519} C_VEL
LIN {X 0,Y 334.415,Z 703.262,A -85,B 0,C 180,E1 13634.269,E2 13634.269} C_VEL
LIN {X 0,Y 335.58,Z 706.609,A -85,B 0,C 180,E1 13633.644,E2 13633.644} C_VEL
LIN {X 0,Y 338.021,Z 711.547,A -85,B 0,C 180,E1 13633.092,E2 13633.092} C_VEL
LIN {X 0,Y 341.373,Z 743.5,A -85,B 0,C 180,E1 13631.624,E2 13631.624} C_VEL
LIN {X 0,Y 341.88,Z 753.337,A -85,B 0,C 180,E1 13631.265,E2 13631.265} C_VEL
LIN {X 0,Y 335.319,Z 907.652,A -85,B 0,C 180,E1 13627.897,E2 13627.897} C_VEL
LIN {X 0,Y 333.493,Z 926.569,A -85,B 0,C 180,E1 13627.219,E2 13627.219} C_VEL
LIN {X 0,Y 330.961,Z 944.31,A -85,B 0,C 180,E1 13626.308,E2 13626.308} C_VEL
LIN {X 0,Y 327.897,Z 961.849,A -85,B 0,C 180,E1 13625.082,E2 13625.082} C_VEL
LIN {X 0,Y 324.52,Z 978.503,A -85,B 0,C 180,E1 13623.576,E2 13623.576} C_VEL
LIN {X 0,Y 320.868,Z 994.834,A -85,B 0,C 180,E1 13621.713,E2 13621.713} C_VEL
LIN {X 0,Y 317.095,Z 1010.621,A -85,B 0,C 180,E1 13619.465,E2 13619.465} C_VEL
LIN {X 0,Y 313.8,Z 1024.102,A -85,B 0,C 180,E1 13617.106,E2 13617.106} C_VEL
LIN {X 0,Y 310.699,Z 1037.133,A -85,B 0,C 180,E1 13614.325,E2 13614.325} C_VEL
LIN {X 0,Y 308.178,Z 1048.68,A -85,B 0,C 180,E1 13611.307,E2 13611.307} C_VEL
LIN {X 0,Y 306.339,Z 1058.742,A -85,B 0,C 180,E1 13608.063,E2 13608.063} C_VEL
LIN {X 0,Y 305.233,Z 1067.261,A -85,B 0,C 180,E1 13604.609,E2 13604.609} C_VEL
LIN {X 0,Y 304.862,Z 1073.802,A -85,B 0,C 180,E1 13601.157,E2 13601.157} C_VEL
LIN {X 0,Y 304.992,Z 1078.511,A -85,B 0,C 180,E1 13597.724,E2 13597.724} C_VEL
LIN {X 0,Y 305.367,Z 1081.443,A -85,B 0,C 180,E1 13594.318,E2 13594.318} C_VEL
LIN {X 0,Y 305.643,Z 1082.537,A -85,B 0,C 180,E1 13591.312,E2 13591.312} C_VEL
LIN {X 0,Y 305.657,Z 1082.237,A -85,B 0,C 180,E1 13588.312,E2 13588.312} C_VEL
LIN {X 0,Y 305.414,Z 1080.519,A -85,B 0,C 180,E1 13585.305,E2 13585.305} C_VEL
LIN {X 0,Y 305.108,Z 1077.084,A -85,B 0,C 180,E1 13582.088,E2 13582.088} C_VEL
LIN {X 0,Y 305.012,Z 1071.568,A -85,B 0,C 180,E1 13578.656,E2 13578.656} C_VEL
LIN {X 0,Y 305.363,Z 1064.516,A -85,B 0,C 180,E1 13575.396,E2 13575.396} C_VEL
LIN {X 0,Y 306.321,Z 1055.468,A -85,B 0,C 180,E1 13572.132,E2 13572.132} C_VEL
LIN {X 0,Y 307.882,Z 1044.878,A -85,B 0,C 180,E1 13569.069,E2 13569.069} C_VEL
LIN {X 0,Y 309.993,Z 1032.798,A -85,B 0,C 180,E1 13566.222,E2 13566.222} C_VEL
LIN {X 0,Y 312.572,Z 1019.167,A -85,B 0,C 180,E1 13563.594,E2 13563.594} C_VEL
LIN {X 0,Y 315.509,Z 1003.957,A -85,B 0,C 180,E1 13561.203,E2 13561.203} C_VEL
LIN {X 0,Y 318.413,Z 988.35,A -85,B 0,C 180,E1 13559.213,E2 13559.213} C_VEL
LIN {X 0,Y 321.349,Z 971.396,A -85,B 0,C 180,E1 13557.479,E2 13557.479} C_VEL
LIN {X 0,Y 324.071,Z 953.523,A -85,B 0,C 180,E1 13556.051,E2 13556.051} C_VEL
LIN {X 0,Y 326.477,Z 934.742,A -85,B 0,C 180,E1 13554.933,E2 13554.933} C_VEL
LIN {X 0,Y 328.247,Z 915.655,A -85,B 0,C 180,E1 13554.141,E2 13554.141} C_VEL
LIN {X 0,Y 329.203,Z 895.005,A -85,B 0,C 180,E1 13553.6,E2 13553.6} C_VEL
LIN {X 0,Y 333.865,Z 748.413,A -85,B 0,C 180,E1 13550.483,E2 13550.483} C_VEL
LIN {X 0,Y 329.606,Z 705.698,A -85,B 0,C 180,E1 13548.918,E2 13548.918} C_VEL
LIN {X 0,Y 329.925,Z 702.223,A -85,B 0,C 180,E1 13548.465,E2 13548.465} C_VEL
LIN {X 0,Y 323.841,Z 682.865,A -85,B 0,C 180,E1 13544.744,E2 13544.744} C_VEL
LIN {X 0,Y 320.857,Z 673.801,A -85,B 0,C 180,E1 13542.791,E2 13542.791} C_VEL
LIN {X 0,Y 320.287,Z 664.291,A -85,B 0,C 180,E1 13539.672,E2 13539.672} C_VEL
LIN {X 0,Y 320.932,Z 658.583,A -85,B 0,C 180,E1 13537.396,E2 13537.396} C_VEL
LIN {X 0,Y 321.387,Z 656.856,A -85,B 0,C 180,E1 13536.614,E2 13536.614} C_VEL
LIN {X 0,Y 321.174,Z 657.131,A -85,B 0,C 180,E1 13534.296,E2 13534.296} C_VEL
LIN {X 0,Y 322.862,Z 660.176,A -85,B 0,C 180,E1 13529.702,E2 13529.702} C_VEL
LIN {X 0,Y 323.315,Z 661.49,A -85,B 0,C 180,E1 13528.844,E2 13528.844} C_VEL
LIN {X 0,Y 325.395,Z 665.678,A -85,B 0,C 180,E1 13526.262,E2 13526.262} C_VEL
LIN {X 0,Y 327.374,Z 670.295,A -85,B 0,C 180,E1 13524.158,E2 13524.158} C_VEL
LIN {X 0,Y 329.842,Z 676.267,A -85,B 0,C 180,E1 13521.891,E2 13521.891} C_VEL
LIN {X 0,Y 332.778,Z 684.913,A -85,B 0,C 180,E1 13519.299,E2 13519.299} C_VEL
LIN {X 0,Y 335.012,Z 693.26,A -85,B 0,C 180,E1 13517.185,E2 13517.185} C_VEL
LIN {X 0,Y 337.057,Z 703.857,A -85,B 0,C 180,E1 13514.912,E2 13514.912} C_VEL
LIN {X 0,Y 333.707,Z 739.375,A -85,B 0,C 180,E1 13510.062,E2 13510.062} C_VEL
LIN {X 0,Y 334.012,Z 742.39,A -85,B 0,C 180,E1 13509.878,E2 13509.878} C_VEL
LIN {X 0,Y 326.523,Z 857.965,A -85,B 0,C 180,E1 13506.439,E2 13506.439} C_VEL
LIN {X 0,Y 325.836,Z 881.461,A -85,B 0,C 180,E1 13505.585,E2 13505.585} C_VEL
LIN {X 0,Y 324.886,Z 897.571,A -85,B 0,C 180,E1 13504.678,E2 13504.678} C_VEL
LIN {X 0,Y 323.419,Z 912.951,A -85,B 0,C 180,E1 13503.471,E2 13503.471} C_VEL
LIN {X 0,Y 321.667,Z 926.922,A -85,B 0,C 180,E1 13502.048,E2 13502.048} C_VEL
LIN {X 0,Y 319.528,Z 940.465,A -85,B 0,C 180,E1 13500.269,E2 13500.269} C_VEL
LIN {X 0,Y 317.387,Z 951.921,A -85,B 0,C 180,E1 13498.375,E2 13498.375} C_VEL
LIN {X 0,Y 314.955,Z 963.228,A -85,B 0,C 180,E1 13495.995,E2 13495.995} C_VEL
LIN {X 0,Y 312.823,Z 972.155,A -85,B 0,C 180,E1 13493.577,E2 13493.577} C_VEL
LIN {X 0,Y 310.873,Z 979.69,A -85,B 0,C 180,E1 13490.899,E2 13490.899} C_VEL
LIN {X 0,Y 309.246,Z 985.439,A -85,B 0,C 180,E1 13488.057,E2 13488.057} C_VEL
LIN {X 0,Y 308.014,Z 989.377,A -85,B 0,C 180,E1 13485.14,E2 13485.14} C_VEL
LIN {X 0,Y 307.162,Z 991.41,A -85,B 0,C 180,E1 13482.182,E2 13482.182} C_VEL
LIN {X 0,Y 306.67,Z 991.687,A -85,B 0,C 180,E1 13479.183,E2 13479.183} C_VEL
LIN {X 0,Y 306.474,Z 990.048,A -85,B 0,C 180,E1 13476.137,E2 13476.137} C_VEL
LIN {X 0,Y 306.58,Z 986.803,A -85,B 0,C 180,E1 13473.252,E2 13473.252} C_VEL
LIN {X 0,Y 306.99,Z 981.606,A -85,B 0,C 180,E1 13470.326,E2 13470.326} C_VEL
LIN {X 0,Y 307.697,Z 974.876,A -85,B 0,C 180,E1 13467.576,E2 13467.576} C_VEL
LIN {X 0,Y 308.746,Z 965.866,A -85,B 0,C 180,E1 13464.799,E2 13464.799} C_VEL
LIN {X 0,Y 309.952,Z 956.093,A -85,B 0,C 180,E1 13462.433,E2 13462.433} C_VEL
LIN {X 0,Y 311.46,Z 943.746,A -85,B 0,C 180,E1 13460.055,E2 13460.055} C_VEL
LIN {X 0,Y 312.911,Z 930.919,A -85,B 0,C 180,E1 13458.1,E2 13458.1} C_VEL
LIN {X 0,Y 314.342,Z 916.555,A -85,B 0,C 180,E1 13456.351,E2 13456.351} C_VEL
LIN {X 0,Y 315.69,Z 900.046,A -85,B 0,C 180,E1 13454.809,E2 13454.809} C_VEL
LIN {X 0,Y 316.665,Z 883.803,A -85,B 0,C 180,E1 13453.692,E2 13453.692} C_VEL
LIN {X 0,Y 317.279,Z 867.004,A -85,B 0,C 180,E1 13452.883,E2 13452.883} C_VEL
LIN {X 0,Y 318.389,Z 821.105,A -85,B 0,C 180,E1 13451.591,E2 13451.591} C_VEL
LIN {X 0,Y 321.74,Z 731.606,A -85,B 0,C 180,E1 13449.193,E2 13449.193} C_VEL
LIN {X 0,Y 320.433,Z 722.528,A -85,B 0,C 180,E1 13448.781,E2 13448.781} C_VEL
LIN {X 0,Y 322.253,Z 690.018,A -85,B 0,C 180,E1 13444.378,E2 13444.378} C_VEL
LIN {X 0,Y 322.095,Z 686.562,A -85,B 0,C 180,E1 13443.864,E2 13443.864} C_VEL
LIN {X 0,Y 317.117,Z 668.241,A -85,B 0,C 180,E1 13440.716,E2 13440.716} C_VEL
LIN {X 0,Y 311.595,Z 651.034,A -85,B 0,C 180,E1 13437.522,E2 13437.522} C_VEL
LIN {X 0,Y 311.591,Z 651.245,A -85,B 0,C 180,E1 13437.186,E2 13437.186} C_VEL
LIN {X 0,Y 315.76,Z 664.322,A -85,B 0,C 180,E1 13433.515,E2 13433.515} C_VEL
LIN {X 0,Y 319.594,Z 678.211,A -85,B 0,C 180,E1 13429.939,E2 13429.939} C_VEL
LIN {X 0,Y 322.938,Z 692.261,A -85,B 0,C 180,E1 13426.596,E2 13426.596} C_VEL
LIN {X 0,Y 322.292,Z 696.924,A -85,B 0,C 180,E1 13425.798,E2 13425.798} C_VEL
LIN {X 0,Y 329.615,Z 737.587,A -85,B 0,C 180,E1 13423.961,E2 13423.961} C_VEL
LIN {X 0,Y 325.749,Z 853.826,A -85,B 0,C 180,E1 13421.374,E2 13421.374} C_VEL
LIN {X 0,Y 324.834,Z 871.173,A -85,B 0,C 180,E1 13420.666,E2 13420.666} C_VEL
LIN {X 0,Y 323.484,Z 887.294,A -85,B 0,C 180,E1 13419.698,E2 13419.698} C_VEL
LIN {X 0,Y 321.664,Z 903.319,A -85,B 0,C 180,E1 13418.401,E2 13418.401} C_VEL
LIN {X 0,Y 319.546,Z 918.133,A -85,B 0,C 180,E1 13416.829,E2 13416.829} C_VEL
LIN {X 0,Y 317.503,Z 930.59,A -85,B 0,C 180,E1 13415.179,E2 13415.179} C_VEL
LIN {X 0,Y 315.556,Z 936.549,A -85,B 0,C 180,E1 13414.344,E2 13414.344} C_VEL
LIN {X 0,Y 308.589,Z 948.533,A -85,B 0,C 180,E1 13412.608,E2 13412.608} C_VEL
LIN {X 0,Y 305.718,Z 954.413,A -85,B 0,C 180,E1 13411.486,E2 13411.486} C_VEL
LIN {X 0,Y 305.331,Z 955.797,A -85,B 0,C 180,E1 13411.169,E2 13411.169} C_VEL
LIN {X 0,Y 303.15,Z 965.957,A -85,B 0,C 180,E1 13408.489,E2 13408.489} C_VEL
LIN {X 0,Y 301.35,Z 974.5,A -85,B 0,C 180,E1 13405.624,E2 13405.624} C_VEL
LIN {X 0,Y 300.028,Z 981.131,A -85,B 0,C 180,E1 13402.725,E2 13402.725} C_VEL
LIN {X 0,Y 299.107,Z 986.326,A -85,B 0,C 180,E1 13399.601,E2 13399.601} C_VEL
LIN {X 0,Y 298.604,Z 990.006,A -85,B 0,C 180,E1 13396.247,E2 13396.247} C_VEL
LIN {X 0,Y 298.539,Z 991.816,A -85,B 0,C 180,E1 13393.06,E2 13393.06} C_VEL
LIN {X 0,Y 298.897,Z 991.936,A -85,B 0,C 180,E1 13389.642,E2 13389.642} C_VEL
LIN {X 0,Y 299.779,Z 990.238,A -85,B 0,C 180,E1 13386.199,E2 13386.199} C_VEL
LIN {X 0,Y 301.169,Z 986.85,A -85,B 0,C 180,E1 13382.946,E2 13382.946} C_VEL
LIN {X 0,Y 303.19,Z 981.477,A -85,B 0,C 180,E1 13379.698,E2 13379.698} C_VEL
LIN {X 0,Y 305.745,Z 974.514,A -85,B 0,C 180,E1 13376.675,E2 13376.675} C_VEL
LIN {X 0,Y 308.719,Z 965.988,A -85,B 0,C 180,E1 13373.883,E2 13373.883} C_VEL
LIN {X 0,Y 311.977,Z 955.912,A -85,B 0,C 180,E1 13371.321,E2 13371.321} C_VEL
LIN {X 0,Y 315.446,Z 944.251,A -85,B 0,C 180,E1 13368.972,E2 13368.972} C_VEL
LIN {X 0,Y 318.804,Z 931.635,A -85,B 0,C 180,E1 13366.95,E2 13366.95} C_VEL
LIN {X 0,Y 321.993,Z 917.651,A -85,B 0,C 180,E1 13365.18,E2 13365.18} C_VEL
LIN {X 0,Y 324.882,Z 902.523,A -85,B 0,C 180,E1 13363.678,E2 13363.678} C_VEL
LIN {X 0,Y 327.284,Z 886.581,A -85,B 0,C 180,E1 13362.467,E2 13362.467} C_VEL
LIN {X 0,Y 329.041,Z 869.678,A -85,B 0,C 180,E1 13361.542,E2 13361.542} C_VEL
LIN {X 0,Y 330.117,Z 851.986,A -85,B 0,C 180,E1 13360.905,E2 13360.905} C_VEL
LIN {X 0,Y 335.071,Z 742.273,A -85,B 0,C 180,E1 13358.411,E2 13358.411} C_VEL
LIN {X 0,Y 329.528,Z 714.412,A -85,B 0,C 180,E1 13356.614,E2 13356.614} C_VEL
LIN {X 0,Y 328.596,Z 711.146,A -85,B 0,C 180,E1 13356.342,E2 13356.342} C_VEL
LIN {X 0,Y 321.302,Z 698.018,A -85,B 0,C 180,E1 13354.498,E2 13354.498} C_VEL
LIN {X 0,Y 318.446,Z 687.438,A -85,B 0,C 180,E1 13351.203,E2 13351.203} C_VEL
LIN {X 0,Y 315.223,Z 677.313,A -85,B 0,C 180,E1 13347.588,E2 13347.588} C_VEL
LIN {X 0,Y 312.338,Z 668.981,A -85,B 0,C 180,E1 13344.17,E2 13344.17} C_VEL
LIN {X 0,Y 309.514,Z 661.848,A -85,B 0,C 180,E1 13340.815,E2 13340.815} C_VEL
LIN {X 0,Y 307.746,Z 657.69,A -85,B 0,C 180,E1 13338.567,E2 13338.567} C_VEL
LIN {X 0,Y 306.429,Z 654.45,A -85,B 0,C 180,E1 13336.687,E2 13336.687} C_VEL
LIN {X 0,Y 304.602,Z 650.371,A -85,B 0,C 180,E1 13334.059,E2 13334.059} C_VEL
LIN {X 0,Y 302.689,Z 646.204,A -85,B 0,C 180,E1 13330.853,E2 13330.853} C_VEL
LIN {X 0,Y 300.444,Z 641.631,A -85,B 0,C 180,E1 13326.305,E2 13326.305} C_VEL
LIN {X 0,Y 298.377,Z 637.576,A -85,B 0,C 180,E1 13319.232,E2 13319.232} C_VEL
LIN {X 0,Y 298.301,Z 637.121,A -85,B 0,C 180,E1 13315.386,E2 13315.386} C_VEL
LIN {X 0,Y 298.325,Z 637.296,A -85,B 0,C 180,E1 13310.937,E2 13310.937} C_VEL
LIN {X 0,Y 298.999,Z 639.489,A -85,B 0,C 180,E1 13306.463,E2 13306.463} C_VEL
LIN {X 0,Y 301.061,Z 642.586,A -85,B 0,C 180,E1 13302.01,E2 13302.01} C_VEL
LIN {X 0,Y 303.679,Z 647.654,A -85,B 0,C 180,E1 13297.547,E2 13297.547} C_VEL
LIN {X 0,Y 306.144,Z 652.606,A -85,B 0,C 180,E1 13294.255,E2 13294.255} C_VEL
LIN {X 0,Y 308.436,Z 657.387,A -85,B 0,C 180,E1 13291.541,E2 13291.541} C_VEL
LIN {X 0,Y 310.628,Z 662.112,A -85,B 0,C 180,E1 13289.217,E2 13289.217} C_VEL
LIN {X 0,Y 313.868,Z 668.933,A -85,B 0,C 180,E1 13286.246,E2 13286.246} C_VEL
LIN {X 0,Y 318.307,Z 679.628,A -85,B 0,C 180,E1 13282.333,E2 13282.333} C_VEL
LIN {X 0,Y 322.777,Z 691.458,A -85,B 0,C 180,E1 13278.715,E2 13278.715} C_VEL
LIN {X 0,Y 326.909,Z 704.007,A -85,B 0,C 180,E1 13275.449,E2 13275.449} C_VEL
LIN {X 0,Y 328.136,Z 706.984,A -85,B 0,C 180,E1 13274.922,E2 13274.922} C_VEL
LIN {X 0,Y 332.528,Z 715.455,A -85,B 0,C 180,E1 13273.888,E2 13273.888} C_VEL
LIN {X 0,Y 335.659,Z 747.505,A -85,B 0,C 180,E1 13272.4,E2 13272.4} C_VEL
LIN {X 0,Y 335.897,Z 754.765,A -85,B 0,C 180,E1 13272.147,E2 13272.147} C_VEL
LIN {X 0,Y 329.087,Z 906.903,A -85,B 0,C 180,E1 13268.775,E2 13268.775} C_VEL
LIN {X 0,Y 327.197,Z 925.784,A -85,B 0,C 180,E1 13268.089,E2 13268.089} C_VEL
LIN {X 0,Y 324.507,Z 943.818,A -85,B 0,C 180,E1 13267.15,E2 13267.15} C_VEL
LIN {X 0,Y 321.32,Z 961.232,A -85,B 0,C 180,E1 13265.913,E2 13265.913} C_VEL
LIN {X 0,Y 317.604,Z 978.659,A -85,B 0,C 180,E1 13264.299,E2 13264.299} C_VEL
LIN {X 0,Y 313.727,Z 995.016,A -85,B 0,C 180,E1 13262.372,E2 13262.372} C_VEL
LIN {X 0,Y 309.913,Z 1010.087,A -85,B 0,C 180,E1 13260.159,E2 13260.159} C_VEL
LIN {X 0,Y 306.266,Z 1024.167,A -85,B 0,C 180,E1 13257.618,E2 13257.618} C_VEL
LIN {X 0,Y 303.022,Z 1037.002,A -85,B 0,C 180,E1 13254.774,E2 13254.774} C_VEL
LIN {X 0,Y 300.377,Z 1048.362,A -85,B 0,C 180,E1 13251.683,E2 13251.683} C_VEL
LIN {X 0,Y 298.44,Z 1058.239,A -85,B 0,C 180,E1 13248.356,E2 13248.356} C_VEL
LIN {X 0,Y 297.277,Z 1066.578,A -85,B 0,C 180,E1 13244.81,E2 13244.81} C_VEL
LIN {X 0,Y 296.887,Z 1072.981,A -85,B 0,C 180,E1 13241.264,E2 13241.264} C_VEL
LIN {X 0,Y 297.038,Z 1077.564,A -85,B 0,C 180,E1 13237.738,E2 13237.738} C_VEL
LIN {X 0,Y 297.42,Z 1080.285,A -85,B 0,C 180,E1 13234.434,E2 13234.434} C_VEL
LIN {X 0,Y 297.727,Z 1081.352,A -85,B 0,C 180,E1 13231.347,E2 13231.347} C_VEL
LIN {X 0,Y 297.746,Z 1081.009,A -85,B 0,C 180,E1 13228.268,E2 13228.268} C_VEL
LIN {X 0,Y 297.484,Z 1079.236,A -85,B 0,C 180,E1 13225.179,E2 13225.179} C_VEL
LIN {X 0,Y 297.154,Z 1075.736,A -85,B 0,C 180,E1 13221.875,E2 13221.875} C_VEL
LIN {X 0,Y 297.055,Z 1070.516,A -85,B 0,C 180,E1 13218.545,E2 13218.545} C_VEL
LIN {X 0,Y 297.468,Z 1062.988,A -85,B 0,C 180,E1 13215,E2 13215} C_VEL
LIN {X 0,Y 298.424,Z 1054.447,A -85,B 0,C 180,E1 13211.844,E2 13211.844} C_VEL
LIN {X 0,Y 300.062,Z 1043.876,A -85,B 0,C 180,E1 13208.702,E2 13208.702} C_VEL
LIN {X 0,Y 302.269,Z 1031.813,A -85,B 0,C 180,E1 13205.784,E2 13205.784} C_VEL
LIN {X 0,Y 304.956,Z 1018.221,A -85,B 0,C 180,E1 13203.098,E2 13203.098} C_VEL
LIN {X 0,Y 308.022,Z 1002.967,A -85,B 0,C 180,E1 13200.649,E2 13200.649} C_VEL
LIN {X 0,Y 311.041,Z 987.333,A -85,B 0,C 180,E1 13198.616,E2 13198.616} C_VEL
LIN {X 0,Y 314.013,Z 970.781,A -85,B 0,C 180,E1 13196.89,E2 13196.89} C_VEL
LIN {X 0,Y 316.745,Z 953.53,A -85,B 0,C 180,E1 13195.476,E2 13195.476} C_VEL
LIN {X 0,Y 319.167,Z 935.496,A -85,B 0,C 180,E1 13194.36,E2 13194.36} C_VEL
LIN {X 0,Y 321.086,Z 916.263,A -85,B 0,C 180,E1 13193.517,E2 13193.517} C_VEL
LIN {X 0,Y 322.11,Z 896.017,A -85,B 0,C 180,E1 13192.96,E2 13192.96} C_VEL
LIN {X 0,Y 326.987,Z 749.264,A -85,B 0,C 180,E1 13189.781,E2 13189.781} C_VEL
LIN {X 0,Y 322.741,Z 705.704,A -85,B 0,C 180,E1 13188.145,E2 13188.145} C_VEL
LIN {X 0,Y 320.054,Z 696.204,A -85,B 0,C 180,E1 13186.337,E2 13186.337} C_VEL
LIN {X 0,Y 317.569,Z 682.413,A -85,B 0,C 180,E1 13182.81,E2 13182.81} C_VEL
LIN {X 0,Y 317.18,Z 671.759,A -85,B 0,C 180,E1 13179.436,E2 13179.436} C_VEL
LIN {X 0,Y 317.973,Z 665.508,A -85,B 0,C 180,E1 13176.912,E2 13176.912} C_VEL
LIN {X 0,Y 318.264,Z 664.18,A -85,B 0,C 180,E1 13176.157,E2 13176.157} C_VEL
LIN {X 0,Y 318.03,Z 664.887,A -85,B 0,C 180,E1 13173.577,E2 13173.577} C_VEL
LIN {X 0,Y 319.555,Z 667.657,A -85,B 0,C 180,E1 13169.559,E2 13169.559} C_VEL
LIN {X 0,Y 321.078,Z 671.554,A -85,B 0,C 180,E1 13167.042,E2 13167.042} C_VEL
LIN {X 0,Y 323.122,Z 676.808,A -85,B 0,C 180,E1 13164.497,E2 13164.497} C_VEL
LIN {X 0,Y 325.514,Z 683.275,A -85,B 0,C 180,E1 13162.008,E2 13162.008} C_VEL
LIN {X 0,Y 328.108,Z 691.872,A -85,B 0,C 180,E1 13159.4,E2 13159.4} C_VEL
LIN {X 0,Y 330.159,Z 700.424,A -85,B 0,C 180,E1 13157.264,E2 13157.264} C_VEL
LIN {X 0,Y 331.383,Z 708.196,A -85,B 0,C 180,E1 13155.577,E2 13155.577} C_VEL
LIN {X 0,Y 327.913,Z 741.066,A -85,B 0,C 180,E1 13151.016,E2 13151.016} C_VEL
LIN {X 0,Y 328.251,Z 744.22,A -85,B 0,C 180,E1 13150.813,E2 13150.813} C_VEL
LIN {X 0,Y 320.31,Z 858.373,A -85,B 0,C 180,E1 13147.33,E2 13147.33} C_VEL
LIN {X 0,Y 319.445,Z 882.996,A -85,B 0,C 180,E1 13146.402,E2 13146.402} C_VEL
LIN {X 0,Y 318.326,Z 900.005,A -85,B 0,C 180,E1 13145.407,E2 13145.407} C_VEL
LIN {X 0,Y 316.674,Z 915.9,A -85,B 0,C 180,E1 13144.108,E2 13144.108} C_VEL
LIN {X 0,Y 314.764,Z 929.604,A -85,B 0,C 180,E1 13142.64,E2 13142.64} C_VEL
LIN {X 0,Y 312.373,Z 943.448,A -85,B 0,C 180,E1 13140.733,E2 13140.733} C_VEL
LIN {X 0,Y 309.996,Z 955.042,A -85,B 0,C 180,E1 13138.706,E2 13138.706} C_VEL
LIN {X 0,Y 307.57,Z 965.526,A -85,B 0,C 180,E1 13136.392,E2 13136.392} C_VEL
LIN {X 0,Y 305.192,Z 974.576,A -85,B 0,C 180,E1 13133.793,E2 13133.793} C_VEL
LIN {X 0,Y 303.306,Z 981.342,A -85,B 0,C 180,E1 13131.278,E2 13131.278} C_VEL
LIN {X 0,Y 301.542,Z 987.047,A -85,B 0,C 180,E1 13128.33,E2 13128.33} C_VEL
LIN {X 0,Y 300.293,Z 990.654,A -85,B 0,C 180,E1 13125.539,E2 13125.539} C_VEL
LIN {X 0,Y 299.351,Z 992.697,A -85,B 0,C 180,E1 13122.505,E2 13122.505} C_VEL
LIN {X 0,Y 298.796,Z 992.982,A -85,B 0,C 180,E1 13119.429,E2 13119.429} C_VEL
LIN {X 0,Y 298.562,Z 991.351,A -85,B 0,C 180,E1 13116.304,E2 13116.304} C_VEL
LIN {X 0,Y 298.649,Z 988.108,A -85,B 0,C 180,E1 13113.344,E2 13113.344} C_VEL
LIN {X 0,Y 299.055,Z 982.921,A -85,B 0,C 180,E1 13110.341,E2 13110.341} C_VEL
LIN {X 0,Y 299.777,Z 976.212,A -85,B 0,C 180,E1 13107.52,E2 13107.52} C_VEL
LIN {X 0,Y 300.852,Z 967.196,A -85,B 0,C 180,E1 13104.67,E2 13104.67} C_VEL
LIN {X 0,Y 302.097,Z 957.442,A -85,B 0,C 180,E1 13102.243,E2 13102.243} C_VEL
LIN {X 0,Y 303.651,Z 945.091,A -85,B 0,C 180,E1 13099.805,E2 13099.805} C_VEL
LIN {X 0,Y 305.178,Z 932.069,A -85,B 0,C 180,E1 13097.77,E2 13097.77} C_VEL
LIN {X 0,Y 306.637,Z 917.97,A -85,B 0,C 180,E1 13096.009,E2 13096.009} C_VEL
LIN {X 0,Y 307.94,Z 902.74,A -85,B 0,C 180,E1 13094.535,E2 13094.535} C_VEL
LIN {X 0,Y 308.981,Z 886.839,A -85,B 0,C 180,E1 13093.371,E2 13093.371} C_VEL
LIN {X 0,Y 309.701,Z 869,A -85,B 0,C 180,E1 13092.46,E2 13092.46} C_VEL
LIN {X 0,Y 310.657,Z 828.305,A -85,B 0,C 180,E1 13091.262,E2 13091.262} C_VEL
LIN {X 0,Y 314.421,Z 732.655,A -85,B 0,C 180,E1 13088.622,E2 13088.622} C_VEL
LIN {X 0,Y 313.129,Z 723.798,A -85,B 0,C 180,E1 13088.231,E2 13088.231} C_VEL
LIN {X 0,Y 315.057,Z 690.909,A -85,B 0,C 180,E1 13083.737,E2 13083.737} C_VEL
LIN {X 0,Y 311.252,Z 675.786,A -85,B 0,C 180,E1 13081.145,E2 13081.145} C_VEL
LIN {X 0,Y 305.749,Z 657.956,A -85,B 0,C 180,E1 13077.882,E2 13077.882} C_VEL
LIN {X 0,Y 305.169,Z 655.905,A -85,B 0,C 180,E1 13077.387,E2 13077.387} C_VEL
LIN {X 0,Y 305.226,Z 656.633,A -85,B 0,C 180,E1 13076.998,E2 13076.998} C_VEL
LIN {X 0,Y 309.146,Z 669.211,A -85,B 0,C 180,E1 13073.442,E2 13073.442} C_VEL
LIN {X 0,Y 312.861,Z 683.086,A -85,B 0,C 180,E1 13069.802,E2 13069.802} C_VEL
LIN {X 0,Y 315.549,Z 694.929,A -85,B 0,C 180,E1 13066.949,E2 13066.949} C_VEL
LIN {X 0,Y 315.3,Z 697.068,A -85,B 0,C 180,E1 13066.607,E2 13066.607} C_VEL
LIN {X 0,Y 322.731,Z 738.706,A -85,B 0,C 180,E1 13064.666,E2 13064.666} C_VEL
LIN {X 0,Y 318.721,Z 854.365,A -85,B 0,C 180,E1 13062.048,E2 13062.048} C_VEL
LIN {X 0,Y 317.783,Z 871.605,A -85,B 0,C 180,E1 13061.336,E2 13061.336} C_VEL
LIN {X 0,Y 316.291,Z 888.689,A -85,B 0,C 180,E1 13060.289,E2 13060.289} C_VEL
LIN {X 0,Y 314.394,Z 904.575,A -85,B 0,C 180,E1 13058.966,E2 13058.966} C_VEL
LIN {X 0,Y 312.191,Z 919.334,A -85,B 0,C 180,E1 13057.361,E2 13057.361} C_VEL
LIN {X 0,Y 309.816,Z 933.155,A -85,B 0,C 180,E1 13055.464,E2 13055.464} C_VEL
LIN {X 0,Y 307.466,Z 945.472,A -85,B 0,C 180,E1 13053.356,E2 13053.356} C_VEL
LIN {X 0,Y 305.331,Z 955.797,A -85,B 0,C 180,E1 13051.169,E2 13051.169} C_VEL
LIN {X 0,Y 303.374,Z 960.596,A -85,B 0,C 180,E1 13050.069,E2 13050.069} C_VEL
LIN {X 0,Y 296.53,Z 969.998,A -85,B 0,C 180,E1 13047.754,E2 13047.754} C_VEL
LIN {X 0,Y 293.899,Z 974.403,A -85,B 0,C 180,E1 13046.351,E2 13046.351} C_VEL
LIN {X 0,Y 293.597,Z 975.413,A -85,B 0,C 180,E1 13045.974,E2 13045.974} C_VEL
LIN {X 0,Y 292.174,Z 982.254,A -85,B 0,C 180,E1 13042.924,E2 13042.924} C_VEL
LIN {X 0,Y 291.21,Z 987.465,A -85,B 0,C 180,E1 13039.716,E2 13039.716} C_VEL
LIN {X 0,Y 290.687,Z 991.164,A -85,B 0,C 180,E1 13036.271,E2 13036.271} C_VEL
LIN {X 0,Y 290.627,Z 993,A -85,B 0,C 180,E1 13032.997,E2 13032.997} C_VEL
LIN {X 0,Y 291.017,Z 993.156,A -85,B 0,C 180,E1 13029.486,E2 13029.486} C_VEL
LIN {X 0,Y 291.963,Z 991.493,A -85,B 0,C 180,E1 13025.951,E2 13025.951} C_VEL
LIN {X 0,Y 293.446,Z 988.158,A -85,B 0,C 180,E1 13022.614,E2 13022.614} C_VEL
LIN {X 0,Y 295.589,Z 982.838,A -85,B 0,C 180,E1 13019.285,E2 13019.285} C_VEL
LIN {X 0,Y 298.285,Z 975.931,A -85,B 0,C 180,E1 13016.191,E2 13016.191} C_VEL
LIN {X 0,Y 301.417,Z 967.515,A -85,B 0,C 180,E1 13013.338,E2 13013.338} C_VEL
LIN {X 0,Y 304.839,Z 957.528,A -85,B 0,C 180,E1 13010.722,E2 13010.722} C_VEL
LIN {X 0,Y 308.588,Z 945.589,A -85,B 0,C 180,E1 13008.254,E2 13008.254} C_VEL
LIN {X 0,Y 312.086,Z 933.14,A -85,B 0,C 180,E1 13006.21,E2 13006.21} C_VEL
LIN {X 0,Y 315.452,Z 919.138,A -85,B 0,C 180,E1 13004.397,E2 13004.397} C_VEL
LIN {X 0,Y 318.548,Z 903.71,A -85,B 0,C 180,E1 13002.834,E2 13002.834} C_VEL
LIN {X 0,Y 321.021,Z 888.137,A -85,B 0,C 180,E1 13001.626,E2 13001.626} C_VEL
LIN {X 0,Y 322.9,Z 871.252,A -85,B 0,C 180,E1 13000.673,E2 13000.673} C_VEL
LIN {X 0,Y 324.074,Z 853.337,A -85,B 0,C 180,E1 13000.007,E2 13000.007} C_VEL
LIN {X 0,Y 329.263,Z 743.887,A -85,B 0,C 180,E1 12997.48,E2 12997.48} C_VEL
LIN {X 0,Y 323.912,Z 716.251,A -85,B 0,C 180,E1 12995.637,E2 12995.637} C_VEL
LIN {X 0,Y 316.515,Z 702.951,A -85,B 0,C 180,E1 12993.724,E2 12993.724} C_VEL
LIN {X 0,Y 313.908,Z 698.535,A -85,B 0,C 180,E1 12993.003,E2 12993.003} C_VEL
LIN {X 0,Y 312.917,Z 695.236,A -85,B 0,C 180,E1 12992.034,E2 12992.034} C_VEL
LIN {X 0,Y 309.822,Z 684.682,A -85,B 0,C 180,E1 12988.321,E2 12988.321} C_VEL
LIN {X 0,Y 306.956,Z 676.116,A -85,B 0,C 180,E1 12984.847,E2 12984.847} C_VEL
LIN {X 0,Y 303.989,Z 667.839,A -85,B 0,C 180,E1 12981.009,E2 12981.009} C_VEL
LIN {X 0,Y 301.788,Z 662.732,A -85,B 0,C 180,E1 12978.146,E2 12978.146} C_VEL
LIN {X 0,Y 300.648,Z 659.865,A -85,B 0,C 180,E1 12976.421,E2 12976.421} C_VEL
LIN {X 0,Y 299.011,Z 656.06,A -85,B 0,C 180,E1 12973.932,E2 12973.932} C_VEL
LIN {X 0,Y 297.196,Z 651.974,A -85,B 0,C 180,E1 12970.664,E2 12970.664} C_VEL
LIN {X 0,Y 295.105,Z 647.577,A -85,B 0,C 180,E1 12966.225,E2 12966.225} C_VEL
LIN {X 0,Y 293.161,Z 643.65,A -85,B 0,C 180,E1 12959.219,E2 12959.219} C_VEL
LIN {X 0,Y 292.821,Z 642.95,A -85,B 0,C 180,E1 12955.3,E2 12955.3} C_VEL
LIN {X 0,Y 293.149,Z 643.434,A -85,B 0,C 180,E1 12950.776,E2 12950.776} C_VEL
LIN {X 0,Y 294.332,Z 646.437,A -85,B 0,C 180,E1 12945.24,E2 12945.24} C_VEL
LIN {X 0,Y 295.925,Z 648.737,A -85,B 0,C 180,E1 12942.094,E2 12942.094} C_VEL
LIN {X 0,Y 298.444,Z 653.772,A -85,B 0,C 180,E1 12937.617,E2 12937.617} C_VEL
LIN {X 0,Y 300.799,Z 658.556,A -85,B 0,C 180,E1 12934.398,E2 12934.398} C_VEL
LIN {X 0,Y 302.962,Z 663.079,A -85,B 0,C 180,E1 12931.783,E2 12931.783} C_VEL
LIN {X 0,Y 305.016,Z 667.658,A -85,B 0,C 180,E1 12929.463,E2 12929.463} C_VEL
LIN {X 0,Y 308.107,Z 674.299,A -85,B 0,C 180,E1 12926.512,E2 12926.512} C_VEL
LIN {X 0,Y 312.46,Z 685.042,A -85,B 0,C 180,E1 12922.521,E2 12922.521} C_VEL
LIN {X 0,Y 316.708,Z 696.52,A -85,B 0,C 180,E1 12918.954,E2 12918.954} C_VEL
LIN {X 0,Y 319.754,Z 705.568,A -85,B 0,C 180,E1 12916.564,E2 12916.564} C_VEL
LIN {X 0,Y 327.062,Z 718.968,A -85,B 0,C 180,E1 12914.733,E2 12914.733} C_VEL
LIN {X 0,Y 329.959,Z 750.907,A -85,B 0,C 180,E1 12913.229,E2 12913.229} C_VEL
LIN {X 0,Y 329.927,Z 757.564,A -85,B 0,C 180,E1 12913.03,E2 12913.03} C_VEL
LIN {X 0,Y 322.971,Z 906.06,A -85,B 0,C 180,E1 12909.695,E2 12909.695} C_VEL
LIN {X 0,Y 321.011,Z 924.912,A -85,B 0,C 180,E1 12909.002,E2 12909.002} C_VEL
LIN {X 0,Y 318.365,Z 942.094,A -85,B 0,C 180,E1 12908.106,E2 12908.106} C_VEL
LIN {X 0,Y 315.023,Z 959.645,A -85,B 0,C 180,E1 12906.86,E2 12906.86} C_VEL
LIN {X 0,Y 311.329,Z 976.346,A -85,B 0,C 180,E1 12905.315,E2 12905.315} C_VEL
LIN {X 0,Y 307.396,Z 992.242,A -85,B 0,C 180,E1 12903.458,E2 12903.458} C_VEL
LIN {X 0,Y 303.257,Z 1007.848,A -85,B 0,C 180,E1 12901.174,E2 12901.174} C_VEL
LIN {X 0,Y 299.524,Z 1021.387,A -85,B 0,C 180,E1 12898.73,E2 12898.73} C_VEL
LIN {X 0,Y 295.978,Z 1034.461,A -85,B 0,C 180,E1 12895.835,E2 12895.835} C_VEL
LIN {X 0,Y 293.047,Z 1046.047,A -85,B 0,C 180,E1 12892.677,E2 12892.677} C_VEL
LIN {X 0,Y 290.84,Z 1056.139,A -85,B 0,C 180,E1 12889.27,E2 12889.27} C_VEL
LIN {X 0,Y 289.47,Z 1064.694,A -85,B 0,C 180,E1 12885.629,E2 12885.629} C_VEL
LIN {X 0,Y 288.927,Z 1071.275,A -85,B 0,C 180,E1 12881.983,E2 12881.983} C_VEL
LIN {X 0,Y 289.023,Z 1076.029,A -85,B 0,C 180,E1 12878.352,E2 12878.352} C_VEL
LIN {X 0,Y 289.449,Z 1079.002,A -85,B 0,C 180,E1 12874.755,E2 12874.755} C_VEL
LIN {X 0,Y 289.8,Z 1080.131,A -85,B 0,C 180,E1 12871.581,E2 12871.581} C_VEL
LIN {X 0,Y 289.843,Z 1079.845,A -85,B 0,C 180,E1 12868.418,E2 12868.418} C_VEL
LIN {X 0,Y 289.57,Z 1078.115,A -85,B 0,C 180,E1 12865.246,E2 12865.246} C_VEL
LIN {X 0,Y 289.213,Z 1074.646,A -85,B 0,C 180,E1 12861.851,E2 12861.851} C_VEL
LIN {X 0,Y 289.101,Z 1069.446,A -85,B 0,C 180,E1 12858.428,E2 12858.428} C_VEL
LIN {X 0,Y 289.529,Z 1061.945,A -85,B 0,C 180,E1 12854.783,E2 12854.783} C_VEL
LIN {X 0,Y 290.618,Z 1052.808,A -85,B 0,C 180,E1 12851.339,E2 12851.339} C_VEL
LIN {X 0,Y 292.391,Z 1042.113,A -85,B 0,C 180,E1 12848.115,E2 12848.115} C_VEL
LIN {X 0,Y 294.743,Z 1029.893,A -85,B 0,C 180,E1 12845.124,E2 12845.124} C_VEL
LIN {X 0,Y 297.591,Z 1016.117,A -85,B 0,C 180,E1 12842.376,E2 12842.376} C_VEL
LIN {X 0,Y 300.697,Z 1001.298,A -85,B 0,C 180,E1 12839.971,E2 12839.971} C_VEL
LIN {X 0,Y 303.86,Z 985.53,A -85,B 0,C 180,E1 12837.898,E2 12837.898} C_VEL
LIN {X 0,Y 306.944,Z 968.886,A -85,B 0,C 180,E1 12836.149,E2 12836.149} C_VEL
LIN {X 0,Y 309.797,Z 951.365,A -85,B 0,C 180,E1 12834.709,E2 12834.709} C_VEL
LIN {X 0,Y 312.331,Z 932.703,A -85,B 0,C 180,E1 12833.571,E2 12833.571} C_VEL
LIN {X 0,Y 314.167,Z 913.767,A -85,B 0,C 180,E1 12832.765,E2 12832.765} C_VEL
LIN {X 0,Y 315.188,Z 892.683,A -85,B 0,C 180,E1 12832.199,E2 12832.199} C_VEL
LIN {X 0,Y 320.134,Z 750.127,A -85,B 0,C 180,E1 12829.058,E2 12829.058} C_VEL
LIN {X 0,Y 316.84,Z 715.025,A -85,B 0,C 180,E1 12827.688,E2 12827.688} C_VEL
LIN {X 0,Y 317.497,Z 708.856,A -85,B 0,C 180,E1 12827.138,E2 12827.138} C_VEL
LIN {X 0,Y 315.517,Z 699.278,A -85,B 0,C 180,E1 12824.965,E2 12824.965} C_VEL
LIN {X 0,Y 314.002,Z 686.315,A -85,B 0,C 180,E1 12821.477,E2 12821.477} C_VEL
LIN {X 0,Y 314.171,Z 677.208,A -85,B 0,C 180,E1 12818.359,E2 12818.359} C_VEL
LIN {X 0,Y 315.095,Z 672.18,A -85,B 0,C 180,E1 12816.293,E2 12816.293} C_VEL
LIN {X 0,Y 315.227,Z 671.565,A -85,B 0,C 180,E1 12815.93,E2 12815.93} C_VEL
LIN {X 0,Y 314.914,Z 672.595,A -85,B 0,C 180,E1 12813.048,E2 12813.048} C_VEL
LIN {X 0,Y 316.06,Z 674.82,A -85,B 0,C 180,E1 12809.78,E2 12809.78} C_VEL
LIN {X 0,Y 317.587,Z 679.49,A -85,B 0,C 180,E1 12806.757,E2 12806.757} C_VEL
LIN {X 0,Y 319.148,Z 683.911,A -85,B 0,C 180,E1 12804.625,E2 12804.625} C_VEL
LIN {X 0,Y 321.118,Z 689.767,A -85,B 0,C 180,E1 12802.325,E2 12802.325} C_VEL
LIN {X 0,Y 323.422,Z 698.267,A -85,B 0,C 180,E1 12799.692,E2 12799.692} C_VEL
LIN {X 0,Y 325.32,Z 707.625,A -85,B 0,C 180,E1 12797.345,E2 12797.345} C_VEL
LIN {X 0,Y 325.877,Z 712.394,A -85,B 0,C 180,E1 12796.304,E2 12796.304} C_VEL
LIN {X 0,Y 322.346,Z 742.69,A -85,B 0,C 180,E1 12792.04,E2 12792.04} C_VEL
LIN {X 0,Y 322.698,Z 746.162,A -85,B 0,C 180,E1 12791.8,E2 12791.8} C_VEL
LIN {X 0,Y 314.174,Z 859.701,A -85,B 0,C 180,E1 12788.233,E2 12788.233} C_VEL
LIN {X 0,Y 313.188,Z 884.804,A -85,B 0,C 180,E1 12787.256,E2 12787.256} C_VEL
LIN {X 0,Y 311.996,Z 901.491,A -85,B 0,C 180,E1 12786.255,E2 12786.255} C_VEL
LIN {X 0,Y 310.286,Z 916.641,A -85,B 0,C 180,E1 12784.991,E2 12784.991} C_VEL
LIN {X 0,Y 308.164,Z 930.896,A -85,B 0,C 180,E1 12783.441,E2 12783.441} C_VEL
LIN {X 0,Y 305.626,Z 944.79,A -85,B 0,C 180,E1 12781.499,E2 12781.499} C_VEL
LIN {X 0,Y 303.076,Z 956.342,A -85,B 0,C 180,E1 12779.433,E2 12779.433} C_VEL
LIN {X 0,Y 300.377,Z 967.15,A -85,B 0,C 180,E1 12776.983,E2 12776.983} C_VEL
LIN {X 0,Y 297.922,Z 975.902,A -85,B 0,C 180,E1 12774.414,E2 12774.414} C_VEL
LIN {X 0,Y 295.73,Z 983.082,A -85,B 0,C 180,E1 12771.64,E2 12771.64} C_VEL
LIN {X 0,Y 293.812,Z 988.771,A -85,B 0,C 180,E1 12768.548,E2 12768.548} C_VEL
LIN {X 0,Y 292.426,Z 992.329,A -85,B 0,C 180,E1 12765.546,E2 12765.546} C_VEL
LIN {X 0,Y 291.446,Z 994.15,A -85,B 0,C 180,E1 12762.428,E2 12762.428} C_VEL
LIN {X 0,Y 290.897,Z 994.23,A -85,B 0,C 180,E1 12759.476,E2 12759.476} C_VEL
LIN {X 0,Y 290.643,Z 992.437,A -85,B 0,C 180,E1 12756.219,E2 12756.219} C_VEL
LIN {X 0,Y 290.731,Z 989.091,A -85,B 0,C 180,E1 12753.222,E2 12753.222} C_VEL
LIN {X 0,Y 291.161,Z 983.765,A -85,B 0,C 180,E1 12750.136,E2 12750.136} C_VEL
LIN {X 0,Y 291.919,Z 976.864,A -85,B 0,C 180,E1 12747.236,E2 12747.236} C_VEL
LIN {X 0,Y 293.069,Z 967.633,A -85,B 0,C 180,E1 12744.291,E2 12744.291} C_VEL
LIN {X 0,Y 294.369,Z 957.699,A -85,B 0,C 180,E1 12741.816,E2 12741.816} C_VEL
LIN {X 0,Y 295.877,Z 946.131,A -85,B 0,C 180,E1 12739.495,E2 12739.495} C_VEL
LIN {X 0,Y 297.468,Z 933.011,A -85,B 0,C 180,E1 12737.402,E2 12737.402} C_VEL
LIN {X 0,Y 298.939,Z 919.319,A -85,B 0,C 180,E1 12735.649,E2 12735.649} C_VEL
LIN {X 0,Y 300.337,Z 903.606,A -85,B 0,C 180,E1 12734.091,E2 12734.091} C_VEL
LIN {X 0,Y 301.398,Z 888.034,A -85,B 0,C 180,E1 12732.923,E2 12732.923} C_VEL
LIN {X 0,Y 302.163,Z 870.127,A -85,B 0,C 180,E1 12731.983,E2 12731.983} C_VEL
LIN {X 0,Y 303.233,Z 827.871,A -85,B 0,C 180,E1 12730.701,E2 12730.701} C_VEL
LIN {X 0,Y 307.082,Z 733.558,A -85,B 0,C 180,E1 12728.032,E2 12728.032} C_VEL
LIN {X 0,Y 305.865,Z 724.286,A -85,B 0,C 180,E1 12727.566,E2 12727.566} C_VEL
LIN {X 0,Y 307.797,Z 692.958,A -85,B 0,C 180,E1 12723.242,E2 12723.242} C_VEL
LIN {X 0,Y 303.234,Z 675.669,A -85,B 0,C 180,E1 12720.189,E2 12720.189} C_VEL
LIN {X 0,Y 298.705,Z 661.057,A -85,B 0,C 180,E1 12717.404,E2 12717.404} C_VEL
LIN {X 0,Y 298.632,Z 661.277,A -85,B 0,C 180,E1 12717.05,E2 12717.05} C_VEL
LIN {X 0,Y 302.537,Z 674.098,A -85,B 0,C 180,E1 12713.366,E2 12713.366} C_VEL
LIN {X 0,Y 306.106,Z 688.035,A -85,B 0,C 180,E1 12709.661,E2 12709.661} C_VEL
LIN {X 0,Y 308.197,Z 697.125,A -85,B 0,C 180,E1 12707.482,E2 12707.482} C_VEL
LIN {X 0,Y 314.918,Z 733.535,A -85,B 0,C 180,E1 12705.679,E2 12705.679} C_VEL
LIN {X 0,Y 315.87,Z 740.469,A -85,B 0,C 180,E1 12705.385,E2 12705.385} C_VEL
LIN {X 0,Y 311.725,Z 854.934,A -85,B 0,C 180,E1 12702.746,E2 12702.746} C_VEL
LIN {X 0,Y 310.755,Z 872.153,A -85,B 0,C 180,E1 12702.025,E2 12702.025} C_VEL
LIN {X 0,Y 309.256,Z 888.757,A -85,B 0,C 180,E1 12700.997,E2 12700.997} C_VEL
LIN {X 0,Y 307.282,Z 904.858,A -85,B 0,C 180,E1 12699.647,E2 12699.647} C_VEL
LIN {X 0,Y 304.971,Z 919.821,A -85,B 0,C 180,E1 12698.001,E2 12698.001} C_VEL
LIN {X 0,Y 302.387,Z 934.275,A -85,B 0,C 180,E1 12695.979,E2 12695.979} C_VEL
LIN {X 0,Y 299.939,Z 946.576,A -85,B 0,C 180,E1 12693.823,E2 12693.823} C_VEL
LIN {X 0,Y 297.495,Z 957.847,A -85,B 0,C 180,E1 12691.349,E2 12691.349} C_VEL
LIN {X 0,Y 295.298,Z 967.698,A -85,B 0,C 180,E1 12688.642,E2 12688.642} C_VEL
LIN {X 0,Y 293.597,Z 975.413,A -85,B 0,C 180,E1 12685.974,E2 12685.974} C_VEL
LIN {X 0,Y 291.945,Z 978.889,A -85,B 0,C 180,E1 12684.653,E2 12684.653} C_VEL
LIN {X 0,Y 286.535,Z 984.599,A -85,B 0,C 180,E1 12682.226,E2 12682.226} C_VEL
LIN {X 0,Y 283.754,Z 987.654,A -85,B 0,C 180,E1 12680.509,E2 12680.509} C_VEL
LIN {X 0,Y 283.295,Z 988.701,A -85,B 0,C 180,E1 12679.757,E2 12679.757} C_VEL
LIN {X 0,Y 282.77,Z 992.32,A -85,B 0,C 180,E1 12676.296,E2 12676.296} C_VEL
LIN {X 0,Y 282.725,Z 994.245,A -85,B 0,C 180,E1 12672.719,E2 12672.719} C_VEL
LIN {X 0,Y 283.182,Z 994.326,A -85,B 0,C 180,E1 12669.108,E2 12669.108} C_VEL
LIN {X 0,Y 284.233,Z 992.605,A -85,B 0,C 180,E1 12665.475,E2 12665.475} C_VEL
LIN {X 0,Y 285.852,Z 989.184,A -85,B 0,C 180,E1 12662.05,E2 12662.05} C_VEL
LIN {X 0,Y 288.174,Z 983.808,A -85,B 0,C 180,E1 12658.638,E2 12658.638} C_VEL
LIN {X 0,Y 291.068,Z 976.851,A -85,B 0,C 180,E1 12655.473,E2 12655.473} C_VEL
LIN {X 0,Y 294.398,Z 968.35,A -85,B 0,C 180,E1 12652.56,E2 12652.56} C_VEL
LIN {X 0,Y 298.019,Z 958.319,A -85,B 0,C 180,E1 12649.898,E2 12649.898} C_VEL
LIN {X 0,Y 301.814,Z 946.825,A -85,B 0,C 180,E1 12647.483,E2 12647.483} C_VEL
LIN {X 0,Y 305.478,Z 934.428,A -85,B 0,C 180,E1 12645.407,E2 12645.407} C_VEL
LIN {X 0,Y 309.029,Z 920.414,A -85,B 0,C 180,E1 12643.553,E2 12643.553} C_VEL
LIN {X 0,Y 312.306,Z 904.877,A -85,B 0,C 180,E1 12641.95,E2 12641.95} C_VEL
LIN {X 0,Y 315.028,Z 888.491,A -85,B 0,C 180,E1 12640.664,E2 12640.664} C_VEL
LIN {X 0,Y 316.962,Z 871.666,A -85,B 0,C 180,E1 12639.713,E2 12639.713} C_VEL
LIN {X 0,Y 318.176,Z 853.85,A -85,B 0,C 180,E1 12639.047,E2 12639.047} C_VEL
LIN {X 0,Y 323.548,Z 745.522,A -85,B 0,C 180,E1 12636.516,E2 12636.516} C_VEL
LIN {X 0,Y 318.857,Z 720.52,A -85,B 0,C 180,E1 12634.8,E2 12634.8} C_VEL
LIN {X 0,Y 311.868,Z 707.963,A -85,B 0,C 180,E1 12632.917,E2 12632.917} C_VEL
LIN {X 0,Y 306.292,Z 698.574,A -85,B 0,C 180,E1 12631.268,E2 12631.268} C_VEL
LIN {X 0,Y 304.702,Z 693.239,A -85,B 0,C 180,E1 12629.487,E2 12629.487} C_VEL
LIN {X 0,Y 301.722,Z 683.707,A -85,B 0,C 180,E1 12625.729,E2 12625.729} C_VEL
LIN {X 0,Y 299.004,Z 675.851,A -85,B 0,C 180,E1 12622.139,E2 12622.139} C_VEL
LIN {X 0,Y 296.556,Z 669.318,A -85,B 0,C 180,E1 12618.665,E2 12618.665} C_VEL
LIN {X 0,Y 294.868,Z 665.268,A -85,B 0,C 180,E1 12616.144,E2 12616.144} C_VEL
LIN {X 0,Y 293.281,Z 661.532,A -85,B 0,C 180,E1 12613.606,E2 12613.606} C_VEL
LIN {X 0,Y 291.703,Z 657.742,A -85,B 0,C 180,E1 12610.467,E2 12610.467} C_VEL
LIN {X 0,Y 289.777,Z 653.533,A -85,B 0,C 180,E1 12606.141,E2 12606.141} C_VEL
LIN {X 0,Y 287.962,Z 649.678,A -85,B 0,C 180,E1 12599.006,E2 12599.006} C_VEL
LIN {X 0,Y 287.716,Z 649.116,A -85,B 0,C 180,E1 12594.816,E2 12594.816} C_VEL
LIN {X 0,Y 288.088,Z 649.689,A -85,B 0,C 180,E1 12590.612,E2 12590.612} C_VEL
LIN {X 0,Y 289.689,Z 653.306,A -85,B 0,C 180,E1 12584.177,E2 12584.177} C_VEL
LIN {X 0,Y 290.769,Z 654.868,A -85,B 0,C 180,E1 12582.18,E2 12582.18} C_VEL
LIN {X 0,Y 293.182,Z 659.787,A -85,B 0,C 180,E1 12577.756,E2 12577.756} C_VEL
LIN {X 0,Y 295.412,Z 664.462,A -85,B 0,C 180,E1 12574.542,E2 12574.542} C_VEL
LIN {X 0,Y 297.523,Z 668.934,A -85,B 0,C 180,E1 12571.935,E2 12571.935} C_VEL
LIN {X 0,Y 299.97,Z 674.495,A -85,B 0,C 180,E1 12569.116,E2 12569.116} C_VEL
LIN {X 0,Y 302.978,Z 681.407,A -85,B 0,C 180,E1 12566.102,E2 12566.102} C_VEL
LIN {X 0,Y 306.668,Z 690.603,A -85,B 0,C 180,E1 12562.668,E2 12562.668} C_VEL
LIN {X 0,Y 310.71,Z 701.81,A -85,B 0,C 180,E1 12559.132,E2 12559.132} C_VEL
LIN {X 0,Y 311.978,Z 705.336,A -85,B 0,C 180,E1 12558.194,E2 12558.194} C_VEL
LIN {X 0,Y 320.273,Z 719.932,A -85,B 0,C 180,E1 12555.972,E2 12555.972} C_VEL
LIN {X 0,Y 321.795,Z 723.321,A -85,B 0,C 180,E1 12555.567,E2 12555.567} C_VEL
LIN {X 0,Y 324.364,Z 754.54,A -85,B 0,C 180,E1 12554.083,E2 12554.083} C_VEL
LIN {X 0,Y 316.944,Z 905.268,A -85,B 0,C 180,E1 12550.65,E2 12550.65} C_VEL
LIN {X 0,Y 314.917,Z 924.074,A -85,B 0,C 180,E1 12549.952,E2 12549.952} C_VEL
LIN {X 0,Y 312.081,Z 941.743,A -85,B 0,C 180,E1 12549.017,E2 12549.017} C_VEL
LIN {X 0,Y 308.602,Z 959.165,A -85,B 0,C 180,E1 12547.759,E2 12547.759} C_VEL
LIN {X 0,Y 304.546,Z 976.576,A -85,B 0,C 180,E1 12546.108,E2 12546.108} C_VEL
LIN {X 0,Y 300.267,Z 992.903,A -85,B 0,C 180,E1 12544.131,E2 12544.131} C_VEL
LIN {X 0,Y 295.966,Z 1008.2,A -85,B 0,C 180,E1 12541.803,E2 12541.803} C_VEL
LIN {X 0,Y 292.078,Z 1021.505,A -85,B 0,C 180,E1 12539.309,E2 12539.309} C_VEL
LIN {X 0,Y 288.373,Z 1034.376,A -85,B 0,C 180,E1 12536.347,E2 12536.347} C_VEL
LIN {X 0,Y 285.299,Z 1045.763,A -85,B 0,C 180,E1 12533.111,E2 12533.111} C_VEL
LIN {X 0,Y 282.975,Z 1055.673,A -85,B 0,C 180,E1 12529.613,E2 12529.613} C_VEL
LIN {X 0,Y 281.527,Z 1064.04,A -85,B 0,C 180,E1 12525.87,E2 12525.87} C_VEL
LIN {X 0,Y 280.956,Z 1070.47,A -85,B 0,C 180,E1 12522.12,E2 12522.12} C_VEL
LIN {X 0,Y 281.065,Z 1075.089,A -85,B 0,C 180,E1 12518.386,E2 12518.386} C_VEL
LIN {X 0,Y 281.503,Z 1077.849,A -85,B 0,C 180,E1 12514.89,E2 12514.89} C_VEL
LIN {X 0,Y 281.883,Z 1078.946,A -85,B 0,C 180,E1 12511.626,E2 12511.626} C_VEL
LIN {X 0,Y 281.94,Z 1078.679,A -85,B 0,C 180,E1 12508.577,E2 12508.577} C_VEL
LIN {X 0,Y 281.657,Z 1076.991,A -85,B 0,C 180,E1 12505.316,E2 12505.316} C_VEL
LIN {X 0,Y 281.271,Z 1073.551,A -85,B 0,C 180,E1 12501.825,E2 12501.825} C_VEL
LIN {X 0,Y 281.146,Z 1068.37,A -85,B 0,C 180,E1 12498.304,E2 12498.304} C_VEL
LIN {X 0,Y 281.55,Z 1061.375,A -85,B 0,C 180,E1 12494.764,E2 12494.764} C_VEL
LIN {X 0,Y 282.65,Z 1052.374,A -85,B 0,C 180,E1 12491.221,E2 12491.221} C_VEL
LIN {X 0,Y 284.463,Z 1041.819,A -85,B 0,C 180,E1 12487.907,E2 12487.907} C_VEL
LIN {X 0,Y 286.879,Z 1029.758,A -85,B 0,C 180,E1 12484.836,E2 12484.836} C_VEL
LIN {X 0,Y 289.806,Z 1016.162,A -85,B 0,C 180,E1 12482.016,E2 12482.016} C_VEL
LIN {X 0,Y 293.138,Z 1000.902,A -85,B 0,C 180,E1 12479.454,E2 12479.454} C_VEL
LIN {X 0,Y 296.41,Z 985.231,A -85,B 0,C 180,E1 12477.335,E2 12477.335} C_VEL
LIN {X 0,Y 299.609,Z 968.612,A -85,B 0,C 180,E1 12475.54,E2 12475.54} C_VEL
LIN {X 0,Y 302.604,Z 950.924,A -85,B 0,C 180,E1 12474.049,E2 12474.049} C_VEL
LIN {X 0,Y 305.145,Z 933.027,A -85,B 0,C 180,E1 12472.921,E2 12472.921} C_VEL
LIN {X 0,Y 307.108,Z 913.818,A -85,B 0,C 180,E1 12472.07,E2 12472.07} C_VEL
LIN {X 0,Y 308.172,Z 893.33,A -85,B 0,C 180,E1 12471.498,E2 12471.498} C_VEL
LIN {X 0,Y 313.336,Z 751.013,A -85,B 0,C 180,E1 12468.305,E2 12468.305} C_VEL
LIN {X 0,Y 311.168,Z 727.748,A -85,B 0,C 180,E1 12467.354,E2 12467.354} C_VEL
LIN {X 0,Y 313.208,Z 713.267,A -85,B 0,C 180,E1 12466.152,E2 12466.152} C_VEL
LIN {X 0,Y 311.673,Z 704.458,A -85,B 0,C 180,E1 12464.06,E2 12464.06} C_VEL
LIN {X 0,Y 310.614,Z 691.867,A -85,B 0,C 180,E1 12460.559,E2 12460.559} C_VEL
LIN {X 0,Y 311.102,Z 683.822,A -85,B 0,C 180,E1 12457.755,E2 12457.755} C_VEL
LIN {X 0,Y 312.148,Z 678.949,A -85,B 0,C 180,E1 12455.722,E2 12455.722} C_VEL
LIN {X 0,Y 311.786,Z 680.358,A -85,B 0,C 180,E1 12452.381,E2 12452.381} C_VEL
LIN {X 0,Y 312.578,Z 682.133,A -85,B 0,C 180,E1 12449.903,E2 12449.903} C_VEL
LIN {X 0,Y 313.825,Z 686.293,A -85,B 0,C 180,E1 12447.103,E2 12447.103} C_VEL
LIN {X 0,Y 315.143,Z 690.594,A -85,B 0,C 180,E1 12444.959,E2 12444.959} C_VEL
LIN {X 0,Y 317.002,Z 696.93,A -85,B 0,C 180,E1 12442.435,E2 12442.435} C_VEL
LIN {X 0,Y 318.981,Z 705.501,A -85,B 0,C 180,E1 12439.787,E2 12439.787} C_VEL
LIN {X 0,Y 320.518,Z 715.39,A -85,B 0,C 180,E1 12437.335,E2 12437.335} C_VEL
LIN {X 0,Y 320.372,Z 718.061,A -85,B 0,C 180,E1 12436.872,E2 12436.872} C_VEL
LIN {X 0,Y 316.957,Z 744.405,A -85,B 0,C 180,E1 12433.105,E2 12433.105} C_VEL
LIN {X 0,Y 317.306,Z 748.122,A -85,B 0,C 180,E1 12432.829,E2 12432.829} C_VEL
LIN {X 0,Y 308.301,Z 859.658,A -85,B 0,C 180,E1 12429.243,E2 12429.243} C_VEL
LIN {X 0,Y 307.128,Z 885.956,A -85,B 0,C 180,E1 12428.197,E2 12428.197} C_VEL
LIN {X 0,Y 305.885,Z 901.82,A -85,B 0,C 180,E1 12427.229,E2 12427.229} C_VEL
LIN {X 0,Y 304.067,Z 917.212,A -85,B 0,C 180,E1 12425.945,E2 12425.945} C_VEL
LIN {X 0,Y 301.818,Z 931.68,A -85,B 0,C 180,E1 12424.369,E2 12424.369} C_VEL
LIN {X 0,Y 299.203,Z 944.981,A -85,B 0,C 180,E1 12422.489,E2 12422.489} C_VEL
LIN {X 0,Y 296.473,Z 956.789,A -85,B 0,C 180,E1 12420.386,E2 12420.386} C_VEL
LIN {X 0,Y 293.727,Z 967.145,A -85,B 0,C 180,E1 12418.049,E2 12418.049} C_VEL
LIN {X 0,Y 291.073,Z 976.068,A -85,B 0,C 180,E1 12415.468,E2 12415.468} C_VEL
LIN {X 0,Y 288.486,Z 983.993,A -85,B 0,C 180,E1 12412.432,E2 12412.432} C_VEL
LIN {X 0,Y 286.528,Z 989.374,A -85,B 0,C 180,E1 12409.545,E2 12409.545} C_VEL
LIN {X 0,Y 284.911,Z 993.278,A -85,B 0,C 180,E1 12406.4,E2 12406.4} C_VEL
LIN {X 0,Y 283.764,Z 995.318,A -85,B 0,C 180,E1 12403.206,E2 12403.206} C_VEL
LIN {X 0,Y 283.063,Z 995.58,A -85,B 0,C 180,E1 12399.962,E2 12399.962} C_VEL
LIN {X 0,Y 282.744,Z 994.08,A -85,B 0,C 180,E1 12396.844,E2 12396.844} C_VEL
LIN {X 0,Y 282.78,Z 990.684,A -85,B 0,C 180,E1 12393.543,E2 12393.543} C_VEL
LIN {X 0,Y 283.137,Z 985.936,A -85,B 0,C 180,E1 12390.602,E2 12390.602} C_VEL
LIN {X 0,Y 283.85,Z 979.331,A -85,B 0,C 180,E1 12387.627,E2 12387.627} C_VEL
LIN {X 0,Y 284.855,Z 971.285,A -85,B 0,C 180,E1 12384.854,E2 12384.854} C_VEL
LIN {X 0,Y 286.245,Z 960.946,A -85,B 0,C 180,E1 12382.064,E2 12382.064} C_VEL
LIN {X 0,Y 287.751,Z 949.732,A -85,B 0,C 180,E1 12379.668,E2 12379.668} C_VEL
LIN {X 0,Y 289.366,Z 937.171,A -85,B 0,C 180,E1 12377.506,E2 12377.506} C_VEL
LIN {X 0,Y 290.918,Z 923.511,A -85,B 0,C 180,E1 12375.634,E2 12375.634} C_VEL
LIN {X 0,Y 292.38,Z 908.633,A -85,B 0,C 180,E1 12374.02,E2 12374.02} C_VEL
LIN {X 0,Y 293.632,Z 891.807,A -85,B 0,C 180,E1 12372.649,E2 12372.649} C_VEL
LIN {X 0,Y 294.458,Z 875.292,A -85,B 0,C 180,E1 12371.691,E2 12371.691} C_VEL
LIN {X 0,Y 294.909,Z 856.014,A -85,B 0,C 180,E1 12370.982,E2 12370.982} C_VEL
LIN {X 0,Y 299.809,Z 734.671,A -85,B 0,C 180,E1 12367.424,E2 12367.424} C_VEL
LIN {X 0,Y 298.598,Z 725.311,A -85,B 0,C 180,E1 12366.946,E2 12366.946} C_VEL
LIN {X 0,Y 300.538,Z 695.445,A -85,B 0,C 180,E1 12362.783,E2 12362.783} C_VEL
LIN {X 0,Y 295.768,Z 677.615,A -85,B 0,C 180,E1 12359.576,E2 12359.576} C_VEL
LIN {X 0,Y 292.248,Z 666.102,A -85,B 0,C 180,E1 12357.343,E2 12357.343} C_VEL
LIN {X 0,Y 292.183,Z 666.336,A -85,B 0,C 180,E1 12356.964,E2 12356.964} C_VEL
LIN {X 0,Y 295.935,Z 679.207,A -85,B 0,C 180,E1 12353.22,E2 12353.22} C_VEL
LIN {X 0,Y 299.531,Z 693.828,A -85,B 0,C 180,E1 12349.298,E2 12349.298} C_VEL
LIN {X 0,Y 300.445,Z 697.486,A -85,B 0,C 180,E1 12348.474,E2 12348.474} C_VEL
LIN {X 0,Y 302.315,Z 702.01,A -85,B 0,C 180,E1 12348.084,E2 12348.084} C_VEL
LIN {X 0,Y 309.095,Z 741.192,A -85,B 0,C 180,E1 12346.159,E2 12346.159} C_VEL
LIN {X 0,Y 304.778,Z 855.501,A -85,B 0,C 180,E1 12343.476,E2 12343.476} C_VEL
LIN {X 0,Y 303.774,Z 872.702,A -85,B 0,C 180,E1 12342.747,E2 12342.747} C_VEL
LIN {X 0,Y 302.134,Z 890.076,A -85,B 0,C 180,E1 12341.647,E2 12341.647} C_VEL
LIN {X 0,Y 300.077,Z 906.061,A -85,B 0,C 180,E1 12340.269,E2 12340.269} C_VEL
LIN {X 0,Y 297.748,Z 920.542,A -85,B 0,C 180,E1 12338.641,E2 12338.641} C_VEL
LIN {X 0,Y 295.099,Z 934.787,A -85,B 0,C 180,E1 12336.616,E2 12336.616} C_VEL
LIN {X 0,Y 292.432,Z 947.672,A -85,B 0,C 180,E1 12334.314,E2 12334.314} C_VEL
LIN {X 0,Y 289.884,Z 958.936,A -85,B 0,C 180,E1 12331.779,E2 12331.779} C_VEL
LIN {X 0,Y 287.59,Z 968.792,A -85,B 0,C 180,E1 12329.004,E2 12329.004} C_VEL
LIN {X 0,Y 285.661,Z 977.23,A -85,B 0,C 180,E1 12325.986,E2 12325.986} C_VEL
LIN {X 0,Y 284.166,Z 984.094,A -85,B 0,C 180,E1 12322.723,E2 12322.723} C_VEL
LIN {X 0,Y 283.295,Z 988.701,A -85,B 0,C 180,E1 12319.757,E2 12319.757} C_VEL
LIN {X 0,Y 282.013,Z 990.651,A -85,B 0,C 180,E1 12318.254,E2 12318.254} C_VEL
LIN {X 0,Y 277.315,Z 993.701,A -85,B 0,C 180,E1 12315.5,E2 12315.5} C_VEL
LIN {X 0,Y 275.044,Z 995.04,A -85,B 0,C 180,E1 12313.606,E2 12313.606} C_VEL
LIN {X 0,Y 274.806,Z 995.381,A -85,B 0,C 180,E1 12312.798,E2 12312.798} C_VEL
LIN {X 0,Y 275.265,Z 995.599,A -85,B 0,C 180,E1 12309.148,E2 12309.148} C_VEL
LIN {X 0,Y 276.347,Z 994.008,A -85,B 0,C 180,E1 12305.413,E2 12305.413} C_VEL
LIN {X 0,Y 278.124,Z 990.586,A -85,B 0,C 180,E1 12301.738,E2 12301.738} C_VEL
LIN {X 0,Y 280.443,Z 985.583,A -85,B 0,C 180,E1 12298.393,E2 12298.393} C_VEL
LIN {X 0,Y 283.441,Z 978.803,A -85,B 0,C 180,E1 12295.148,E2 12295.148} C_VEL
LIN {X 0,Y 286.897,Z 970.548,A -85,B 0,C 180,E1 12292.167,E2 12292.167} C_VEL
LIN {X 0,Y 290.656,Z 960.842,A -85,B 0,C 180,E1 12289.447,E2 12289.447} C_VEL
LIN {X 0,Y 294.581,Z 949.66,A -85,B 0,C 180,E1 12286.983,E2 12286.983} C_VEL
LIN {X 0,Y 298.556,Z 937.012,A -85,B 0,C 180,E1 12284.767,E2 12284.767} C_VEL
LIN {X 0,Y 302.243,Z 923.545,A -85,B 0,C 180,E1 12282.892,E2 12282.892} C_VEL
LIN {X 0,Y 305.529,Z 909.168,A -85,B 0,C 180,E1 12281.319,E2 12281.319} C_VEL
LIN {X 0,Y 308.387,Z 893.531,A -85,B 0,C 180,E1 12280,E2 12280} C_VEL
LIN {X 0,Y 310.669,Z 876.564,A -85,B 0,C 180,E1 12278.937,E2 12278.937} C_VEL
LIN {X 0,Y 312.112,Z 859.471,A -85,B 0,C 180,E1 12278.207,E2 12278.207} C_VEL
LIN {X 0,Y 315.738,Z 790.155,A -85,B 0,C 180,E1 12276.517,E2 12276.517} C_VEL
LIN {X 0,Y 317.939,Z 747.075,A -85,B 0,C 180,E1 12275.508,E2 12275.508} C_VEL
LIN {X 0,Y 313.81,Z 724.611,A -85,B 0,C 180,E1 12273.917,E2 12273.917} C_VEL
LIN {X 0,Y 305.299,Z 709.385,A -85,B 0,C 180,E1 12271.492,E2 12271.492} C_VEL
LIN {X 0,Y 298.836,Z 698.962,A -85,B 0,C 180,E1 12269.462,E2 12269.462} C_VEL
LIN {X 0,Y 296.827,Z 692.487,A -85,B 0,C 180,E1 12267.049,E2 12267.049} C_VEL
LIN {X 0,Y 294.025,Z 683.803,A -85,B 0,C 180,E1 12263.233,E2 12263.233} C_VEL
LIN {X 0,Y 291.626,Z 677.211,A -85,B 0,C 180,E1 12259.842,E2 12259.842} C_VEL
LIN {X 0,Y 289.534,Z 671.453,A -85,B 0,C 180,E1 12256.45,E2 12256.45} C_VEL
LIN {X 0,Y 287.731,Z 667.252,A -85,B 0,C 180,E1 12253.464,E2 12253.464} C_VEL
LIN {X 0,Y 286.183,Z 663.482,A -85,B 0,C 180,E1 12250.264,E2 12250.264} C_VEL
LIN {X 0,Y 284.466,Z 659.503,A -85,B 0,C 180,E1 12246.053,E2 12246.053} C_VEL
LIN {X 0,Y 282.788,Z 655.785,A -85,B 0,C 180,E1 12238.987,E2 12238.987} C_VEL
LIN {X 0,Y 282.622,Z 655.282,A -85,B 0,C 180,E1 12234.926,E2 12234.926} C_VEL
LIN {X 0,Y 282.972,Z 655.843,A -85,B 0,C 180,E1 12230.646,E2 12230.646} C_VEL
LIN {X 0,Y 284.631,Z 659.529,A -85,B 0,C 180,E1 12224.098,E2 12224.098} C_VEL
LIN {X 0,Y 285.58,Z 661.002,A -85,B 0,C 180,E1 12222.233,E2 12222.233} C_VEL
LIN {X 0,Y 287.896,Z 665.697,A -85,B 0,C 180,E1 12217.971,E2 12217.971} C_VEL
LIN {X 0,Y 290.03,Z 670.364,A -85,B 0,C 180,E1 12214.693,E2 12214.693} C_VEL
LIN {X 0,Y 292.102,Z 674.885,A -85,B 0,C 180,E1 12212.021,E2 12212.021} C_VEL
LIN {X 0,Y 295.183,Z 681.699,A -85,B 0,C 180,E1 12208.558,E2 12208.558} C_VEL
LIN {X 0,Y 298.961,Z 691.09,A -85,B 0,C 180,E1 12204.649,E2 12204.649} C_VEL
LIN {X 0,Y 302.939,Z 701.874,A -85,B 0,C 180,E1 12200.921,E2 12200.921} C_VEL
LIN {X 0,Y 304.397,Z 705.549,A -85,B 0,C 180,E1 12199.894,E2 12199.894} C_VEL
LIN {X 0,Y 312.343,Z 718.975,A -85,B 0,C 180,E1 12197.605,E2 12197.605} C_VEL
LIN {X 0,Y 316.52,Z 726.978,A -85,B 0,C 180,E1 12196.47,E2 12196.47} C_VEL
LIN {X 0,Y 318.697,Z 755.922,A -85,B 0,C 180,E1 12195.071,E2 12195.071} C_VEL
LIN {X 0,Y 311.028,Z 904.485,A -85,B 0,C 180,E1 12191.646,E2 12191.646} C_VEL
LIN {X 0,Y 308.928,Z 923.232,A -85,B 0,C 180,E1 12190.943,E2 12190.943} C_VEL
LIN {X 0,Y 305.88,Z 941.423,A -85,B 0,C 180,E1 12189.964,E2 12189.964} C_VEL
LIN {X 0,Y 302.136,Z 959.243,A -85,B 0,C 180,E1 12188.649,E2 12188.649} C_VEL
LIN {X 0,Y 297.989,Z 976.185,A -85,B 0,C 180,E1 12187.006,E2 12187.006} C_VEL
LIN {X 0,Y 293.566,Z 992.247,A -85,B 0,C 180,E1 12185.022,E2 12185.022} C_VEL
LIN {X 0,Y 289.151,Z 1007.126,A -85,B 0,C 180,E1 12182.716,E2 12182.716} C_VEL
LIN {X 0,Y 284.952,Z 1020.688,A -85,B 0,C 180,E1 12180.116,E2 12180.116} C_VEL
LIN {X 0,Y 281.024,Z 1033.487,A -85,B 0,C 180,E1 12177.091,E2 12177.091} C_VEL
LIN {X 0,Y 277.742,Z 1044.826,A -85,B 0,C 180,E1 12173.778,E2 12173.778} C_VEL
LIN {X 0,Y 275.239,Z 1054.67,A -85,B 0,C 180,E1 12170.188,E2 12170.188} C_VEL
LIN {X 0,Y 273.65,Z 1062.977,A -85,B 0,C 180,E1 12166.34,E2 12166.34} C_VEL
